LIN {X 0,Y 487.957,Z 631.751,A -85,B 0,C 180,E1 -6386.696,E2 -6386.696} C_VEL
LIN {X 0,Y 487.888,Z 633.791,A -85,B 0,C 180,E1 -6388.348,E2 -6388.348} C_VEL
LIN {X 0,Y 487.818,Z 634.497,A -85,B 0,C 180,E1 -6389.999,E2 -6389.999} C_VEL
LIN {X 0,Y 487.886,Z 633.877,A -85,B 0,C 180,E1 -6391.65,E2 -6391.65} C_VEL
LIN {X 0,Y 487.955,Z 631.916,A -85,B 0,C 180,E1 -6393.302,E2 -6393.302} C_VEL
LIN {X 0,Y 487.963,Z 628.565,A -85,B 0,C 180,E1 -6394.956,E2 -6394.956} C_VEL
LIN {X 0,Y 488.052,Z 624.185,A -85,B 0,C 180,E1 -6396.48,E2 -6396.48} C_VEL
LIN {X 0,Y 488.192,Z 619.062,A -85,B 0,C 180,E1 -6397.859,E2 -6397.859} C_VEL
LIN {X 0,Y 488.465,Z 612.281,A -85,B 0,C 180,E1 -6399.314,E2 -6399.314} C_VEL
LIN {X 0,Y 488.822,Z 603.853,A -85,B 0,C 180,E1 -6400.771,E2 -6400.771} C_VEL
LIN {X 0,Y 489.247,Z 594.601,A -85,B 0,C 180,E1 -6402.081,E2 -6402.081} C_VEL
LIN {X 0,Y 489.717,Z 584.411,A -85,B 0,C 180,E1 -6403.273,E2 -6403.273} C_VEL
LIN {X 0,Y 490.248,Z 573.643,A -85,B 0,C 180,E1 -6404.316,E2 -6404.316} C_VEL
LIN {X 0,Y 490.821,Z 561.869,A -85,B 0,C 180,E1 -6405.253,E2 -6405.253} C_VEL
LIN {X 0,Y 491.354,Z 548.87,A -85,B 0,C 180,E1 -6406.088,E2 -6406.088} C_VEL
LIN {X 0,Y 491.917,Z 535.085,A -85,B 0,C 180,E1 -6406.769,E2 -6406.769} C_VEL
LIN {X 0,Y 492.27,Z 521.352,A -85,B 0,C 180,E1 -6407.27,E2 -6407.27} C_VEL
LIN {X 0,Y 492.606,Z 506.72,A -85,B 0,C 180,E1 -6407.62,E2 -6407.62} C_VEL
LIN {X 0,Y 493.536,Z 388.715,A -85,B 0,C 180,E1 -6409.371,E2 -6409.371} C_VEL
LIN {X 0,Y 490.364,Z 372.401,A -85,B 0,C 180,E1 -6409.769,E2 -6409.769} C_VEL
LIN {X 0,Y 490.626,Z 364.751,A -85,B 0,C 180,E1 -6410.983,E2 -6410.983} C_VEL
LIN {X 0,Y 491.223,Z 351.672,A -85,B 0,C 180,E1 -6413.168,E2 -6413.168} C_VEL
LIN {X 0,Y 490.46,Z 346.443,A -85,B 0,C 180,E1 -6414.102,E2 -6414.102} C_VEL
LIN {X 0,Y 488.842,Z 338.631,A -85,B 0,C 180,E1 -6415.549,E2 -6415.549} C_VEL
LIN {X 0,Y 488.781,Z 338.212,A -85,B 0,C 180,E1 -6415.781,E2 -6415.781} C_VEL
LIN {X 0,Y 488.735,Z 338.214,A -85,B 0,C 180,E1 -6418.696,E2 -6418.696} C_VEL
LIN {X 0,Y 488.694,Z 338.234,A -85,B 0,C 180,E1 -6421.178,E2 -6421.178} C_VEL
LIN {X 0,Y 488.732,Z 338.235,A -85,B 0,C 180,E1 -6424.111,E2 -6424.111} C_VEL
LIN {X 0,Y 488.679,Z 338.234,A -85,B 0,C 180,E1 -6427.157,E2 -6427.157} C_VEL
LIN {X 0,Y 488.744,Z 338.225,A -85,B 0,C 180,E1 -6429.248,E2 -6429.248} C_VEL
LIN {X 0,Y 488.726,Z 338.23,A -85,B 0,C 180,E1 -6432.52,E2 -6432.52} C_VEL
LIN {X 0,Y 488.705,Z 338.222,A -85,B 0,C 180,E1 -6435.198,E2 -6435.198} C_VEL
LIN {X 0,Y 488.727,Z 338.229,A -85,B 0,C 180,E1 -6437.478,E2 -6437.478} C_VEL
LIN {X 0,Y 488.741,Z 338.22,A -85,B 0,C 180,E1 -6440.749,E2 -6440.749} C_VEL
LIN {X 0,Y 488.678,Z 338.232,A -85,B 0,C 180,E1 -6443.868,E2 -6443.868} C_VEL
LIN {X 0,Y 488.731,Z 338.229,A -85,B 0,C 180,E1 -6446.876,E2 -6446.876} C_VEL
LIN {X 0,Y 488.725,Z 338.215,A -85,B 0,C 180,E1 -6449.781,E2 -6449.781} C_VEL
LIN {X 0,Y 488.789,Z 338.211,A -85,B 0,C 180,E1 -6453.054,E2 -6453.054} C_VEL
LIN {X 0,Y 488.692,Z 338.233,A -85,B 0,C 180,E1 -6456.254,E2 -6456.254} C_VEL
LIN {X 0,Y 488.737,Z 338.225,A -85,B 0,C 180,E1 -6459.175,E2 -6459.175} C_VEL
LIN {X 0,Y 488.748,Z 338.229,A -85,B 0,C 180,E1 -6461.627,E2 -6461.627} C_VEL
LIN {X 0,Y 488.754,Z 338.221,A -85,B 0,C 180,E1 -6464.999,E2 -6464.999} C_VEL
LIN {X 0,Y 488.822,Z 338.215,A -85,B 0,C 180,E1 -6468.388,E2 -6468.388} C_VEL
LIN {X 0,Y 488.809,Z 338.217,A -85,B 0,C 180,E1 -6471.733,E2 -6471.733} C_VEL
LIN {X 0,Y 488.852,Z 338.211,A -85,B 0,C 180,E1 -6474.224,E2 -6474.224} C_VEL
LIN {X 0,Y 488.953,Z 338.199,A -85,B 0,C 180,E1 -6477.529,E2 -6477.529} C_VEL
LIN {X 0,Y 488.959,Z 338.199,A -85,B 0,C 180,E1 -6480,E2 -6480} C_VEL
LIN {X 0,Y 488.953,Z 338.199,A -85,B 0,C 180,E1 -6482.471,E2 -6482.471} C_VEL
LIN {X 0,Y 488.853,Z 338.212,A -85,B 0,C 180,E1 -6485.776,E2 -6485.776} C_VEL
LIN {X 0,Y 488.808,Z 338.217,A -85,B 0,C 180,E1 -6488.266,E2 -6488.266} C_VEL
LIN {X 0,Y 488.821,Z 338.214,A -85,B 0,C 180,E1 -6491.612,E2 -6491.612} C_VEL
LIN {X 0,Y 488.754,Z 338.221,A -85,B 0,C 180,E1 -6495.001,E2 -6495.001} C_VEL
LIN {X 0,Y 488.744,Z 338.229,A -85,B 0,C 180,E1 -6498.443,E2 -6498.443} C_VEL
LIN {X 0,Y 488.702,Z 338.228,A -85,B 0,C 180,E1 -6501.071,E2 -6501.071} C_VEL
LIN {X 0,Y 488.691,Z 338.232,A -85,B 0,C 180,E1 -6503.746,E2 -6503.746} C_VEL
LIN {X 0,Y 488.789,Z 338.211,A -85,B 0,C 180,E1 -6506.946,E2 -6506.946} C_VEL
LIN {X 0,Y 488.7,Z 338.219,A -85,B 0,C 180,E1 -6510.364,E2 -6510.364} C_VEL
LIN {X 0,Y 488.727,Z 338.228,A -85,B 0,C 180,E1 -6513.485,E2 -6513.485} C_VEL
LIN {X 0,Y 488.681,Z 338.228,A -85,B 0,C 180,E1 -6516.357,E2 -6516.357} C_VEL
LIN {X 0,Y 488.734,Z 338.22,A -85,B 0,C 180,E1 -6519.251,E2 -6519.251} C_VEL
LIN {X 0,Y 488.727,Z 338.229,A -85,B 0,C 180,E1 -6522.522,E2 -6522.522} C_VEL
LIN {X 0,Y 488.705,Z 338.221,A -85,B 0,C 180,E1 -6525.2,E2 -6525.2} C_VEL
LIN {X 0,Y 488.725,Z 338.23,A -85,B 0,C 180,E1 -6527.48,E2 -6527.48} C_VEL
LIN {X 0,Y 488.743,Z 338.225,A -85,B 0,C 180,E1 -6530.752,E2 -6530.752} C_VEL
LIN {X 0,Y 488.681,Z 338.235,A -85,B 0,C 180,E1 -6533.87,E2 -6533.87} C_VEL
LIN {X 0,Y 488.735,Z 338.225,A -85,B 0,C 180,E1 -6536.879,E2 -6536.879} C_VEL
LIN {X 0,Y 488.731,Z 338.223,A -85,B 0,C 180,E1 -6539.783,E2 -6539.783} C_VEL
LIN {X 0,Y 488.796,Z 338.225,A -85,B 0,C 180,E1 -6543.056,E2 -6543.056} C_VEL
LIN {X 0,Y 488.813,Z 338.303,A -85,B 0,C 180,E1 -6544.392,E2 -6544.392} C_VEL
LIN {X 0,Y 491.086,Z 349.656,A -85,B 0,C 180,E1 -6546.526,E2 -6546.526} C_VEL
LIN {X 0,Y 491.009,Z 356.638,A -85,B 0,C 180,E1 -6547.711,E2 -6547.711} C_VEL
LIN {X 0,Y 490.34,Z 372.125,A -85,B 0,C 180,E1 -6550.257,E2 -6550.257} C_VEL
LIN {X 0,Y 491.847,Z 380.023,A -85,B 0,C 180,E1 -6550.473,E2 -6550.473} C_VEL
LIN {X 0,Y 493.591,Z 389.526,A -85,B 0,C 180,E1 -6550.689,E2 -6550.689} C_VEL
LIN {X 0,Y 492.541,Z 509.938,A -85,B 0,C 180,E1 -6552.485,E2 -6552.485} C_VEL
LIN {X 0,Y 492.18,Z 524.147,A -85,B 0,C 180,E1 -6552.864,E2 -6552.864} C_VEL
LIN {X 0,Y 491.837,Z 537.72,A -85,B 0,C 180,E1 -6553.395,E2 -6553.395} C_VEL
LIN {X 0,Y 491.344,Z 549.891,A -85,B 0,C 180,E1 -6554.019,E2 -6554.019} C_VEL
LIN {X 0,Y 490.785,Z 562.69,A -85,B 0,C 180,E1 -6554.852,E2 -6554.852} C_VEL
LIN {X 0,Y 490.242,Z 574.318,A -85,B 0,C 180,E1 -6555.79,E2 -6555.79} C_VEL
LIN {X 0,Y 489.611,Z 585.946,A -85,B 0,C 180,E1 -6556.935,E2 -6556.935} C_VEL
LIN {X 0,Y 489.247,Z 595.237,A -85,B 0,C 180,E1 -6558.046,E2 -6558.046} C_VEL
LIN {X 0,Y 488.842,Z 603.563,A -85,B 0,C 180,E1 -6559.229,E2 -6559.229} C_VEL
LIN {X 0,Y 488.459,Z 612.04,A -85,B 0,C 180,E1 -6560.686,E2 -6560.686} C_VEL
LIN {X 0,Y 488.191,Z 618.866,A -85,B 0,C 180,E1 -6562.141,E2 -6562.141} C_VEL
LIN {X 0,Y 488.039,Z 624.895,A -85,B 0,C 180,E1 -6563.778,E2 -6563.778} C_VEL
LIN {X 0,Y 487.962,Z 628.449,A -85,B 0,C 180,E1 -6565.044,E2 -6565.044} C_VEL
LIN {X 0,Y 487.955,Z 631.837,A -85,B 0,C 180,E1 -6566.698,E2 -6566.698} C_VEL
LIN {X 0,Y 487.885,Z 633.838,A -85,B 0,C 180,E1 -6568.35,E2 -6568.35} C_VEL
LIN {X 0,Y 487.817,Z 634.5,A -85,B 0,C 180,E1 -6570.001,E2 -6570.001} C_VEL
LIN {X 0,Y 487.886,Z 633.834,A -85,B 0,C 180,E1 -6571.652,E2 -6571.652} C_VEL
LIN {X 0,Y 487.956,Z 631.83,A -85,B 0,C 180,E1 -6573.304,E2 -6573.304} C_VEL
LIN {X 0,Y 487.963,Z 628.441,A -85,B 0,C 180,E1 -6574.958,E2 -6574.958} C_VEL
LIN {X 0,Y 488.049,Z 624.037,A -85,B 0,C 180,E1 -6576.479,E2 -6576.479} C_VEL
LIN {X 0,Y 488.194,Z 618.859,A -85,B 0,C 180,E1 -6577.861,E2 -6577.861} C_VEL
LIN {X 0,Y 488.461,Z 612.028,A -85,B 0,C 180,E1 -6579.316,E2 -6579.316} C_VEL
LIN {X 0,Y 488.843,Z 603.549,A -85,B 0,C 180,E1 -6580.773,E2 -6580.773} C_VEL
LIN {X 0,Y 489.255,Z 594.224,A -85,B 0,C 180,E1 -6582.084,E2 -6582.084} C_VEL
LIN {X 0,Y 489.708,Z 583.976,A -85,B 0,C 180,E1 -6583.276,E2 -6583.276} C_VEL
LIN {X 0,Y 490.273,Z 573.121,A -85,B 0,C 180,E1 -6584.317,E2 -6584.317} C_VEL
LIN {X 0,Y 490.881,Z 561.232,A -85,B 0,C 180,E1 -6585.254,E2 -6585.254} C_VEL
LIN {X 0,Y 491.441,Z 548.081,A -85,B 0,C 180,E1 -6586.087,E2 -6586.087} C_VEL
LIN {X 0,Y 491.913,Z 534.836,A -85,B 0,C 180,E1 -6586.735,E2 -6586.735} C_VEL
LIN {X 0,Y 492.258,Z 520.818,A -85,B 0,C 180,E1 -6587.241,E2 -6587.241} C_VEL
LIN {X 0,Y 492.586,Z 507.071,A -85,B 0,C 180,E1 -6587.57,E2 -6587.57} C_VEL
LIN {X 0,Y 493.533,Z 389.002,A -85,B 0,C 180,E1 -6589.321,E2 -6589.321} C_VEL
LIN {X 0,Y 490.329,Z 372.216,A -85,B 0,C 180,E1 -6589.735,E2 -6589.735} C_VEL
LIN {X 0,Y 491.033,Z 355.31,A -85,B 0,C 180,E1 -6592.512,E2 -6592.512} C_VEL
LIN {X 0,Y 491.089,Z 349.648,A -85,B 0,C 180,E1 -6593.474,E2 -6593.474} C_VEL
LIN {X 0,Y 488.815,Z 338.438,A -85,B 0,C 180,E1 -6595.553,E2 -6595.553} C_VEL
LIN {X 0,Y 488.751,Z 338.231,A -85,B 0,C 180,E1 -6597.397,E2 -6597.397} C_VEL
LIN {X 0,Y 488.714,Z 338.236,A -85,B 0,C 180,E1 -6600.364,E2 -6600.364} C_VEL
LIN {X 0,Y 488.741,Z 338.229,A -85,B 0,C 180,E1 -6603.485,E2 -6603.485} C_VEL
LIN {X 0,Y 488.694,Z 338.238,A -85,B 0,C 180,E1 -6606.356,E2 -6606.356} C_VEL
LIN {X 0,Y 488.705,Z 338.233,A -85,B 0,C 180,E1 -6609.255,E2 -6609.255} C_VEL
LIN {X 0,Y 488.711,Z 338.234,A -85,B 0,C 180,E1 -6611.6,E2 -6611.6} C_VEL
LIN {X 0,Y 488.706,Z 338.231,A -85,B 0,C 180,E1 -6614.803,E2 -6614.803} C_VEL
LIN {X 0,Y 488.696,Z 338.237,A -85,B 0,C 180,E1 -6617.475,E2 -6617.475} C_VEL
LIN {X 0,Y 488.738,Z 338.233,A -85,B 0,C 180,E1 -6619.677,E2 -6619.677} C_VEL
LIN {X 0,Y 488.684,Z 338.236,A -85,B 0,C 180,E1 -6622.841,E2 -6622.841} C_VEL
LIN {X 0,Y 488.735,Z 338.234,A -85,B 0,C 180,E1 -6625.888,E2 -6625.888} C_VEL
LIN {X 0,Y 488.697,Z 338.236,A -85,B 0,C 180,E1 -6628.821,E2 -6628.821} C_VEL
LIN {X 0,Y 488.756,Z 338.232,A -85,B 0,C 180,E1 -6632.139,E2 -6632.139} C_VEL
LIN {X 0,Y 488.815,Z 338.538,A -85,B 0,C 180,E1 -6632.646,E2 -6632.646} C_VEL
LIN {X 0,Y 491.201,Z 350.219,A -85,B 0,C 180,E1 -6634.343,E2 -6634.343} C_VEL
LIN {X 0,Y 491.062,Z 365.26,A -85,B 0,C 180,E1 -6636.343,E2 -6636.343} C_VEL
LIN {X 0,Y 490.501,Z 386.847,A -85,B 0,C 180,E1 -6639.23,E2 -6639.23} C_VEL
LIN {X 0,Y 490.05,Z 409.49,A -85,B 0,C 180,E1 -6642.257,E2 -6642.257} C_VEL
LIN {X 0,Y 489.773,Z 420.832,A -85,B 0,C 180,E1 -6643.762,E2 -6643.762} C_VEL
LIN {X 0,Y 491.649,Z 435.316,A -85,B 0,C 180,E1 -6644.106,E2 -6644.106} C_VEL
LIN {X 0,Y 490.761,Z 532.213,A -85,B 0,C 180,E1 -6645.698,E2 -6645.698} C_VEL
LIN {X 0,Y 490.493,Z 544.73,A -85,B 0,C 180,E1 -6646.061,E2 -6646.061} C_VEL
LIN {X 0,Y 490.174,Z 557.03,A -85,B 0,C 180,E1 -6646.58,E2 -6646.58} C_VEL
LIN {X 0,Y 489.83,Z 569.483,A -85,B 0,C 180,E1 -6647.281,E2 -6647.281} C_VEL
LIN {X 0,Y 489.49,Z 580.545,A -85,B 0,C 180,E1 -6648.089,E2 -6648.089} C_VEL
LIN {X 0,Y 489.108,Z 590.871,A -85,B 0,C 180,E1 -6649.025,E2 -6649.025} C_VEL
LIN {X 0,Y 488.755,Z 600.216,A -85,B 0,C 180,E1 -6650.064,E2 -6650.064} C_VEL
LIN {X 0,Y 488.471,Z 609.197,A -85,B 0,C 180,E1 -6651.311,E2 -6651.311} C_VEL
LIN {X 0,Y 488.206,Z 616.433,A -85,B 0,C 180,E1 -6652.556,E2 -6652.556} C_VEL
LIN {X 0,Y 488.063,Z 622.035,A -85,B 0,C 180,E1 -6653.759,E2 -6653.759} C_VEL
LIN {X 0,Y 487.97,Z 626.714,A -85,B 0,C 180,E1 -6655.043,E2 -6655.043} C_VEL
LIN {X 0,Y 487.94,Z 629.073,A -85,B 0,C 180,E1 -6655.87,E2 -6655.87} C_VEL
LIN {X 0,Y 487.967,Z 631.002,A -85,B 0,C 180,E1 -6656.697,E2 -6656.697} C_VEL
LIN {X 0,Y 487.888,Z 632.494,A -85,B 0,C 180,E1 -6657.523,E2 -6657.523} C_VEL
LIN {X 0,Y 487.89,Z 633.528,A -85,B 0,C 180,E1 -6658.349,E2 -6658.349} C_VEL
LIN {X 0,Y 487.82,Z 634.417,A -85,B 0,C 180,E1 -6660,E2 -6660} C_VEL
LIN {X 0,Y 487.834,Z 634.223,A -85,B 0,C 180,E1 -6660.826,E2 -6660.826} C_VEL
LIN {X 0,Y 487.889,Z 633.621,A -85,B 0,C 180,E1 -6661.651,E2 -6661.651} C_VEL
LIN {X 0,Y 487.888,Z 632.625,A -85,B 0,C 180,E1 -6662.477,E2 -6662.477} C_VEL
LIN {X 0,Y 487.967,Z 631.209,A -85,B 0,C 180,E1 -6663.303,E2 -6663.303} C_VEL
LIN {X 0,Y 487.931,Z 628.245,A -85,B 0,C 180,E1 -6664.544,E2 -6664.544} C_VEL
LIN {X 0,Y 488.073,Z 624.216,A -85,B 0,C 180,E1 -6665.785,E2 -6665.785} C_VEL
LIN {X 0,Y 488.186,Z 618.005,A -85,B 0,C 180,E1 -6667.237,E2 -6667.237} C_VEL
LIN {X 0,Y 488.419,Z 611.228,A -85,B 0,C 180,E1 -6668.482,E2 -6668.482} C_VEL
LIN {X 0,Y 488.675,Z 602.725,A -85,B 0,C 180,E1 -6669.729,E2 -6669.729} C_VEL
LIN {X 0,Y 488.979,Z 594.009,A -85,B 0,C 180,E1 -6670.769,E2 -6670.769} C_VEL
LIN {X 0,Y 489.467,Z 583.309,A -85,B 0,C 180,E1 -6671.807,E2 -6671.807} C_VEL
LIN {X 0,Y 489.783,Z 572.519,A -85,B 0,C 180,E1 -6672.643,E2 -6672.643} C_VEL
LIN {X 0,Y 490.141,Z 560.667,A -85,B 0,C 180,E1 -6673.369,E2 -6673.369} C_VEL
LIN {X 0,Y 490.479,Z 548.288,A -85,B 0,C 180,E1 -6673.94,E2 -6673.94} C_VEL
LIN {X 0,Y 490.813,Z 534.532,A -85,B 0,C 180,E1 -6674.38,E2 -6674.38} C_VEL
LIN {X 0,Y 490.944,Z 519.124,A -85,B 0,C 180,E1 -6674.667,E2 -6674.667} C_VEL
LIN {X 0,Y 491.526,Z 433.033,A -85,B 0,C 180,E1 -6676.033,E2 -6676.033} C_VEL
LIN {X 0,Y 489.765,Z 420.903,A -85,B 0,C 180,E1 -6676.318,E2 -6676.318} C_VEL
LIN {X 0,Y 490.41,Z 396.325,A -85,B 0,C 180,E1 -6679.681,E2 -6679.681} C_VEL
LIN {X 0,Y 491.082,Z 374.245,A -85,B 0,C 180,E1 -6682.731,E2 -6682.731} C_VEL
LIN {X 0,Y 491.695,Z 353.431,A -85,B 0,C 180,E1 -6685.621,E2 -6685.621} C_VEL
LIN {X 0,Y 490.347,Z 345.54,A -85,B 0,C 180,E1 -6686.796,E2 -6686.796} C_VEL
LIN {X 0,Y 488.786,Z 338.35,A -85,B 0,C 180,E1 -6687.918,E2 -6687.918} C_VEL
LIN {X 0,Y 488.697,Z 338.235,A -85,B 0,C 180,E1 -6691.18,E2 -6691.18} C_VEL
LIN {X 0,Y 488.736,Z 338.233,A -85,B 0,C 180,E1 -6694.113,E2 -6694.113} C_VEL
LIN {X 0,Y 488.684,Z 338.234,A -85,B 0,C 180,E1 -6697.159,E2 -6697.159} C_VEL
LIN {X 0,Y 488.724,Z 338.235,A -85,B 0,C 180,E1 -6700.344,E2 -6700.344} C_VEL
LIN {X 0,Y 488.689,Z 338.232,A -85,B 0,C 180,E1 -6703.654,E2 -6703.654} C_VEL
LIN {X 0,Y 488.705,Z 338.222,A -85,B 0,C 180,E1 -6704.878,E2 -6704.878} C_VEL
LIN {X 0,Y 488.034,Z 338.306,A -85,B 0,C 180,E1 -6705.566,E2 -6705.566} C_VEL
LIN {X 0,Y 485.172,Z 338.674,A -85,B 0,C 180,E1 -6706.682,E2 -6706.682} C_VEL
LIN {X 0,Y 482.757,Z 338.978,A -85,B 0,C 180,E1 -6707.581,E2 -6707.581} C_VEL
LIN {X 0,Y 481.726,Z 339.105,A -85,B 0,C 180,E1 -6708.276,E2 -6708.276} C_VEL
LIN {X 0,Y 481.646,Z 339.112,A -85,B 0,C 180,E1 -6708.511,E2 -6708.511} C_VEL
LIN {X 0,Y 481.676,Z 339.104,A -85,B 0,C 180,E1 -6711.14,E2 -6711.14} C_VEL
LIN {X 0,Y 481.673,Z 339.107,A -85,B 0,C 180,E1 -6714.794,E2 -6714.794} C_VEL
LIN {X 0,Y 481.677,Z 339.106,A -85,B 0,C 180,E1 -6717.325,E2 -6717.325} C_VEL
LIN {X 0,Y 481.684,Z 339.093,A -85,B 0,C 180,E1 -6720.258,E2 -6720.258} C_VEL
LIN {X 0,Y 481.751,Z 339.101,A -85,B 0,C 180,E1 -6723.112,E2 -6723.112} C_VEL
LIN {X 0,Y 481.765,Z 339.248,A -85,B 0,C 180,E1 -6724.227,E2 -6724.227} C_VEL
LIN {X 0,Y 484.235,Z 351.61,A -85,B 0,C 180,E1 -6726.56,E2 -6726.56} C_VEL
LIN {X 0,Y 483.73,Z 365.505,A -85,B 0,C 180,E1 -6728.924,E2 -6728.924} C_VEL
LIN {X 0,Y 483.415,Z 372.218,A -85,B 0,C 180,E1 -6730.016,E2 -6730.016} C_VEL
LIN {X 0,Y 486.762,Z 389.518,A -85,B 0,C 180,E1 -6730.453,E2 -6730.453} C_VEL
LIN {X 0,Y 485.93,Z 499.574,A -85,B 0,C 180,E1 -6732.1,E2 -6732.1} C_VEL
LIN {X 0,Y 485.686,Z 515.129,A -85,B 0,C 180,E1 -6732.398,E2 -6732.398} C_VEL
LIN {X 0,Y 485.31,Z 528.714,A -85,B 0,C 180,E1 -6732.822,E2 -6732.822} C_VEL
LIN {X 0,Y 484.842,Z 542.31,A -85,B 0,C 180,E1 -6733.418,E2 -6733.418} C_VEL
LIN {X 0,Y 484.262,Z 555.958,A -85,B 0,C 180,E1 -6734.209,E2 -6734.209} C_VEL
LIN {X 0,Y 483.564,Z 568.872,A -85,B 0,C 180,E1 -6735.157,E2 -6735.157} C_VEL
LIN {X 0,Y 482.965,Z 580.493,A -85,B 0,C 180,E1 -6736.214,E2 -6736.214} C_VEL
LIN {X 0,Y 482.406,Z 591.008,A -85,B 0,C 180,E1 -6737.376,E2 -6737.376} C_VEL
LIN {X 0,Y 481.979,Z 600.501,A -85,B 0,C 180,E1 -6738.646,E2 -6738.646} C_VEL
LIN {X 0,Y 481.554,Z 609.56,A -85,B 0,C 180,E1 -6740.125,E2 -6740.125} C_VEL
LIN {X 0,Y 481.242,Z 616.857,A -85,B 0,C 180,E1 -6741.602,E2 -6741.602} C_VEL
LIN {X 0,Y 480.999,Z 623.414,A -85,B 0,C 180,E1 -6743.286,E2 -6743.286} C_VEL
LIN {X 0,Y 480.898,Z 628.327,A -85,B 0,C 180,E1 -6744.968,E2 -6744.968} C_VEL
LIN {X 0,Y 480.88,Z 631.752,A -85,B 0,C 180,E1 -6746.648,E2 -6746.648} C_VEL
LIN {X 0,Y 480.789,Z 633.792,A -85,B 0,C 180,E1 -6748.324,E2 -6748.324} C_VEL
LIN {X 0,Y 480.742,Z 634.497,A -85,B 0,C 180,E1 -6749.999,E2 -6749.999} C_VEL
LIN {X 0,Y 480.787,Z 633.876,A -85,B 0,C 180,E1 -6751.674,E2 -6751.674} C_VEL
LIN {X 0,Y 480.879,Z 631.915,A -85,B 0,C 180,E1 -6753.35,E2 -6753.35} C_VEL
LIN {X 0,Y 480.897,Z 628.563,A -85,B 0,C 180,E1 -6755.029,E2 -6755.029} C_VEL
LIN {X 0,Y 480.997,Z 623.723,A -85,B 0,C 180,E1 -6756.712,E2 -6756.712} C_VEL
LIN {X 0,Y 481.23,Z 617.251,A -85,B 0,C 180,E1 -6758.396,E2 -6758.396} C_VEL
LIN {X 0,Y 481.506,Z 610.046,A -85,B 0,C 180,E1 -6759.874,E2 -6759.874} C_VEL
LIN {X 0,Y 481.948,Z 601.134,A -85,B 0,C 180,E1 -6761.352,E2 -6761.352} C_VEL
LIN {X 0,Y 482.433,Z 591.777,A -85,B 0,C 180,E1 -6762.621,E2 -6762.621} C_VEL
LIN {X 0,Y 482.937,Z 581.412,A -85,B 0,C 180,E1 -6763.785,E2 -6763.785} C_VEL
LIN {X 0,Y 483.513,Z 569.982,A -85,B 0,C 180,E1 -6764.843,E2 -6764.843} C_VEL
LIN {X 0,Y 484.16,Z 557.317,A -85,B 0,C 180,E1 -6765.792,E2 -6765.792} C_VEL
LIN {X 0,Y 484.722,Z 544.996,A -85,B 0,C 180,E1 -6766.53,E2 -6766.53} C_VEL
LIN {X 0,Y 485.193,Z 531.363,A -85,B 0,C 180,E1 -6767.164,E2 -6767.164} C_VEL
LIN {X 0,Y 485.631,Z 517.184,A -85,B 0,C 180,E1 -6767.637,E2 -6767.637} C_VEL
LIN {X 0,Y 485.887,Z 503.683,A -85,B 0,C 180,E1 -6767.926,E2 -6767.926} C_VEL
LIN {X 0,Y 486.829,Z 389.653,A -85,B 0,C 180,E1 -6769.634,E2 -6769.634} C_VEL
LIN {X 0,Y 483.481,Z 372.451,A -85,B 0,C 180,E1 -6770.059,E2 -6770.059} C_VEL
LIN {X 0,Y 483.637,Z 367.364,A -85,B 0,C 180,E1 -6770.855,E2 -6770.855} C_VEL
LIN {X 0,Y 484.274,Z 352.055,A -85,B 0,C 180,E1 -6773.453,E2 -6773.453} C_VEL
LIN {X 0,Y 481.853,Z 339.681,A -85,B 0,C 180,E1 -6775.755,E2 -6775.755} C_VEL
LIN {X 0,Y 481.733,Z 339.118,A -85,B 0,C 180,E1 -6775.954,E2 -6775.954} C_VEL
LIN {X 0,Y 481.683,Z 339.09,A -85,B 0,C 180,E1 -6778.904,E2 -6778.904} C_VEL
LIN {X 0,Y 481.657,Z 339.111,A -85,B 0,C 180,E1 -6782.189,E2 -6782.189} C_VEL
LIN {X 0,Y 481.69,Z 339.106,A -85,B 0,C 180,E1 -6784.68,E2 -6784.68} C_VEL
LIN {X 0,Y 481.657,Z 339.116,A -85,B 0,C 180,E1 -6788.007,E2 -6788.007} C_VEL
LIN {X 0,Y 481.68,Z 339.104,A -85,B 0,C 180,E1 -6790.649,E2 -6790.649} C_VEL
LIN {X 0,Y 481.677,Z 339.108,A -85,B 0,C 180,E1 -6793.294,E2 -6793.294} C_VEL
LIN {X 0,Y 481.683,Z 339.102,A -85,B 0,C 180,E1 -6796.845,E2 -6796.845} C_VEL
LIN {X 0,Y 481.686,Z 339.103,A -85,B 0,C 180,E1 -6800.06,E2 -6800.06} C_VEL
LIN {X 0,Y 481.621,Z 339.101,A -85,B 0,C 180,E1 -6803.252,E2 -6803.252} C_VEL
LIN {X 0,Y 481.701,Z 339.105,A -85,B 0,C 180,E1 -6806.329,E2 -6806.329} C_VEL
LIN {X 0,Y 481.65,Z 339.101,A -85,B 0,C 180,E1 -6809.415,E2 -6809.415} C_VEL
LIN {X 0,Y 481.694,Z 339.093,A -85,B 0,C 180,E1 -6812.168,E2 -6812.168} C_VEL
LIN {X 0,Y 481.71,Z 339.102,A -85,B 0,C 180,E1 -6814.969,E2 -6814.969} C_VEL
LIN {X 0,Y 481.65,Z 339.109,A -85,B 0,C 180,E1 -6817.705,E2 -6817.705} C_VEL
LIN {X 0,Y 481.698,Z 339.102,A -85,B 0,C 180,E1 -6820.393,E2 -6820.393} C_VEL
LIN {X 0,Y 481.682,Z 339.109,A -85,B 0,C 180,E1 -6823.034,E2 -6823.034} C_VEL
LIN {X 0,Y 481.684,Z 339.107,A -85,B 0,C 180,E1 -6825.638,E2 -6825.638} C_VEL
LIN {X 0,Y 481.786,Z 339.091,A -85,B 0,C 180,E1 -6828.216,E2 -6828.216} C_VEL
LIN {X 0,Y 481.754,Z 339.097,A -85,B 0,C 180,E1 -6831.611,E2 -6831.611} C_VEL
LIN {X 0,Y 481.812,Z 339.088,A -85,B 0,C 180,E1 -6834.139,E2 -6834.139} C_VEL
LIN {X 0,Y 481.92,Z 339.076,A -85,B 0,C 180,E1 -6837.492,E2 -6837.492} C_VEL
LIN {X 0,Y 481.93,Z 339.075,A -85,B 0,C 180,E1 -6840,E2 -6840} C_VEL
LIN {X 0,Y 481.92,Z 339.075,A -85,B 0,C 180,E1 -6842.507,E2 -6842.507} C_VEL
LIN {X 0,Y 481.812,Z 339.088,A -85,B 0,C 180,E1 -6845.86,E2 -6845.86} C_VEL
LIN {X 0,Y 481.754,Z 339.096,A -85,B 0,C 180,E1 -6848.388,E2 -6848.388} C_VEL
LIN {X 0,Y 481.785,Z 339.09,A -85,B 0,C 180,E1 -6851.784,E2 -6851.784} C_VEL
LIN {X 0,Y 481.733,Z 339.093,A -85,B 0,C 180,E1 -6855.224,E2 -6855.224} C_VEL
LIN {X 0,Y 481.702,Z 339.108,A -85,B 0,C 180,E1 -6858.722,E2 -6858.722} C_VEL
LIN {X 0,Y 481.644,Z 339.105,A -85,B 0,C 180,E1 -6861.395,E2 -6861.395} C_VEL
LIN {X 0,Y 481.672,Z 339.109,A -85,B 0,C 180,E1 -6864.113,E2 -6864.113} C_VEL
LIN {X 0,Y 481.742,Z 339.087,A -85,B 0,C 180,E1 -6867.141,E2 -6867.141} C_VEL
LIN {X 0,Y 481.669,Z 339.087,A -85,B 0,C 180,E1 -6869.742,E2 -6869.742} C_VEL
LIN {X 0,Y 481.664,Z 339.113,A -85,B 0,C 180,E1 -6872.675,E2 -6872.675} C_VEL
LIN {X 0,Y 481.634,Z 339.11,A -85,B 0,C 180,E1 -6875.71,E2 -6875.71} C_VEL
LIN {X 0,Y 481.706,Z 339.096,A -85,B 0,C 180,E1 -6879.355,E2 -6879.355} C_VEL
LIN {X 0,Y 481.668,Z 339.114,A -85,B 0,C 180,E1 -6882.159,E2 -6882.159} C_VEL
LIN {X 0,Y 481.653,Z 339.101,A -85,B 0,C 180,E1 -6884.458,E2 -6884.458} C_VEL
LIN {X 0,Y 481.681,Z 339.107,A -85,B 0,C 180,E1 -6886.847,E2 -6886.847} C_VEL
LIN {X 0,Y 481.687,Z 339.103,A -85,B 0,C 180,E1 -6890.062,E2 -6890.062} C_VEL
LIN {X 0,Y 481.625,Z 339.113,A -85,B 0,C 180,E1 -6893.255,E2 -6893.255} C_VEL
LIN {X 0,Y 481.704,Z 339.104,A -85,B 0,C 180,E1 -6896.331,E2 -6896.331} C_VEL
LIN {X 0,Y 481.655,Z 339.112,A -85,B 0,C 180,E1 -6899.417,E2 -6899.417} C_VEL
LIN {X 0,Y 481.7,Z 339.103,A -85,B 0,C 180,E1 -6902.17,E2 -6902.17} C_VEL
LIN {X 0,Y 481.748,Z 339.162,A -85,B 0,C 180,E1 -6904.136,E2 -6904.136} C_VEL
LIN {X 0,Y 482.952,Z 344.873,A -85,B 0,C 180,E1 -6905.269,E2 -6905.269} C_VEL
LIN {X 0,Y 484.322,Z 352.933,A -85,B 0,C 180,E1 -6906.746,E2 -6906.746} C_VEL
LIN {X 0,Y 483.425,Z 372.023,A -85,B 0,C 180,E1 -6909.952,E2 -6909.952} C_VEL
LIN {X 0,Y 484.269,Z 376.511,A -85,B 0,C 180,E1 -6910.1,E2 -6910.1} C_VEL
LIN {X 0,Y 486.857,Z 389.883,A -85,B 0,C 180,E1 -6910.416,E2 -6910.416} C_VEL
LIN {X 0,Y 485.785,Z 509.946,A -85,B 0,C 180,E1 -6912.233,E2 -6912.233} C_VEL
LIN {X 0,Y 485.394,Z 524.487,A -85,B 0,C 180,E1 -6912.629,E2 -6912.629} C_VEL
LIN {X 0,Y 484.992,Z 538.853,A -85,B 0,C 180,E1 -6913.208,E2 -6913.208} C_VEL
LIN {X 0,Y 484.441,Z 551.66,A -85,B 0,C 180,E1 -6913.893,E2 -6913.893} C_VEL
LIN {X 0,Y 483.829,Z 564.118,A -85,B 0,C 180,E1 -6914.736,E2 -6914.736} C_VEL
LIN {X 0,Y 483.19,Z 576.663,A -85,B 0,C 180,E1 -6915.793,E2 -6915.793} C_VEL
LIN {X 0,Y 482.568,Z 587.841,A -85,B 0,C 180,E1 -6916.955,E2 -6916.955} C_VEL
LIN {X 0,Y 482.139,Z 597.86,A -85,B 0,C 180,E1 -6918.226,E2 -6918.226} C_VEL
LIN {X 0,Y 481.69,Z 606.18,A -85,B 0,C 180,E1 -6919.493,E2 -6919.493} C_VEL
LIN {X 0,Y 481.326,Z 614.132,A -85,B 0,C 180,E1 -6920.97,E2 -6920.97} C_VEL
LIN {X 0,Y 481.053,Z 620.53,A -85,B 0,C 180,E1 -6922.446,E2 -6922.446} C_VEL
LIN {X 0,Y 480.952,Z 626.204,A -85,B 0,C 180,E1 -6924.13,E2 -6924.13} C_VEL
LIN {X 0,Y 480.816,Z 630.322,A -85,B 0,C 180,E1 -6925.81,E2 -6925.81} C_VEL
LIN {X 0,Y 480.879,Z 631.837,A -85,B 0,C 180,E1 -6926.65,E2 -6926.65} C_VEL
LIN {X 0,Y 480.786,Z 633.838,A -85,B 0,C 180,E1 -6928.326,E2 -6928.326} C_VEL
LIN {X 0,Y 480.741,Z 634.5,A -85,B 0,C 180,E1 -6930.001,E2 -6930.001} C_VEL
LIN {X 0,Y 480.787,Z 633.834,A -85,B 0,C 180,E1 -6931.676,E2 -6931.676} C_VEL
LIN {X 0,Y 480.88,Z 631.83,A -85,B 0,C 180,E1 -6933.352,E2 -6933.352} C_VEL
LIN {X 0,Y 480.897,Z 628.441,A -85,B 0,C 180,E1 -6935.032,E2 -6935.032} C_VEL
LIN {X 0,Y 480.998,Z 623.565,A -85,B 0,C 180,E1 -6936.714,E2 -6936.714} C_VEL
LIN {X 0,Y 481.232,Z 617.05,A -85,B 0,C 180,E1 -6938.399,E2 -6938.399} C_VEL
LIN {X 0,Y 481.522,Z 609.797,A -85,B 0,C 180,E1 -6939.876,E2 -6939.876} C_VEL
LIN {X 0,Y 481.976,Z 600.815,A -85,B 0,C 180,E1 -6941.354,E2 -6941.354} C_VEL
LIN {X 0,Y 482.407,Z 591.383,A -85,B 0,C 180,E1 -6942.624,E2 -6942.624} C_VEL
LIN {X 0,Y 482.951,Z 580.941,A -85,B 0,C 180,E1 -6943.787,E2 -6943.787} C_VEL
LIN {X 0,Y 483.57,Z 569.411,A -85,B 0,C 180,E1 -6944.843,E2 -6944.843} C_VEL
LIN {X 0,Y 484.212,Z 556.617,A -85,B 0,C 180,E1 -6945.793,E2 -6945.793} C_VEL
LIN {X 0,Y 484.71,Z 544.128,A -85,B 0,C 180,E1 -6946.533,E2 -6946.533} C_VEL
LIN {X 0,Y 485.22,Z 531.003,A -85,B 0,C 180,E1 -6947.133,E2 -6947.133} C_VEL
LIN {X 0,Y 485.617,Z 517.779,A -85,B 0,C 180,E1 -6947.574,E2 -6947.574} C_VEL
LIN {X 0,Y 485.834,Z 504.051,A -85,B 0,C 180,E1 -6947.876,E2 -6947.876} C_VEL
LIN {X 0,Y 486.854,Z 390.543,A -85,B 0,C 180,E1 -6949.573,E2 -6949.573} C_VEL
LIN {X 0,Y 483.468,Z 372.591,A -85,B 0,C 180,E1 -6950.005,E2 -6950.005} C_VEL
LIN {X 0,Y 483.466,Z 370.871,A -85,B 0,C 180,E1 -6950.22,E2 -6950.22} C_VEL
LIN {X 0,Y 484.302,Z 352.912,A -85,B 0,C 180,E1 -6953.256,E2 -6953.256} C_VEL
LIN {X 0,Y 482.969,Z 344.846,A -85,B 0,C 180,E1 -6954.732,E2 -6954.732} C_VEL
LIN {X 0,Y 481.805,Z 339.393,A -85,B 0,C 180,E1 -6955.774,E2 -6955.774} C_VEL
LIN {X 0,Y 481.724,Z 339.096,A -85,B 0,C 180,E1 -6955.957,E2 -6955.957} C_VEL
LIN {X 0,Y 481.683,Z 339.095,A -85,B 0,C 180,E1 -6958.904,E2 -6958.904} C_VEL
LIN {X 0,Y 481.661,Z 339.116,A -85,B 0,C 180,E1 -6962.19,E2 -6962.19} C_VEL
LIN {X 0,Y 481.698,Z 339.107,A -85,B 0,C 180,E1 -6964.682,E2 -6964.682} C_VEL
LIN {X 0,Y 481.661,Z 339.114,A -85,B 0,C 180,E1 -6968.008,E2 -6968.008} C_VEL
LIN {X 0,Y 481.661,Z 339.109,A -85,B 0,C 180,E1 -6971.042,E2 -6971.042} C_VEL
LIN {X 0,Y 481.659,Z 339.111,A -85,B 0,C 180,E1 -6974.458,E2 -6974.458} C_VEL
LIN {X 0,Y 481.652,Z 339.115,A -85,B 0,C 180,E1 -6977.84,E2 -6977.84} C_VEL
LIN {X 0,Y 481.684,Z 339.107,A -85,B 0,C 180,E1 -6980.652,E2 -6980.652} C_VEL
LIN {X 0,Y 481.632,Z 339.118,A -85,B 0,C 180,E1 -6983.377,E2 -6983.377} C_VEL
LIN {X 0,Y 481.715,Z 339.106,A -85,B 0,C 180,E1 -6986.33,E2 -6986.33} C_VEL
LIN {X 0,Y 481.655,Z 339.116,A -85,B 0,C 180,E1 -6989.418,E2 -6989.418} C_VEL
LIN {X 0,Y 481.77,Z 339.27,A -85,B 0,C 180,E1 -6992.327,E2 -6992.327} C_VEL
LIN {X 0,Y 484.092,Z 350.058,A -85,B 0,C 180,E1 -6993.95,E2 -6993.95} C_VEL
LIN {X 0,Y 484.488,Z 355.178,A -85,B 0,C 180,E1 -6994.664,E2 -6994.664} C_VEL
LIN {X 0,Y 483.913,Z 379.969,A -85,B 0,C 180,E1 -6997.998,E2 -6997.998} C_VEL
LIN {X 0,Y 483.2,Z 404.701,A -85,B 0,C 180,E1 -7001.338,E2 -7001.338} C_VEL
LIN {X 0,Y 482.85,Z 420.811,A -85,B 0,C 180,E1 -7003.508,E2 -7003.508} C_VEL
LIN {X 0,Y 484.853,Z 436.091,A -85,B 0,C 180,E1 -7003.88,E2 -7003.88} C_VEL
LIN {X 0,Y 483.864,Z 531.429,A -85,B 0,C 180,E1 -7005.49,E2 -7005.49} C_VEL
LIN {X 0,Y 483.591,Z 544.231,A -85,B 0,C 180,E1 -7005.857,E2 -7005.857} C_VEL
LIN {X 0,Y 483.261,Z 556.641,A -85,B 0,C 180,E1 -7006.384,E2 -7006.384} C_VEL
LIN {X 0,Y 482.88,Z 569.273,A -85,B 0,C 180,E1 -7007.102,E2 -7007.102} C_VEL
LIN {X 0,Y 482.504,Z 580.282,A -85,B 0,C 180,E1 -7007.914,E2 -7007.914} C_VEL
LIN {X 0,Y 482.112,Z 590.645,A -85,B 0,C 180,E1 -7008.863,E2 -7008.863} C_VEL
LIN {X 0,Y 481.715,Z 600.03,A -85,B 0,C 180,E1 -7009.917,E2 -7009.917} C_VEL
LIN {X 0,Y 481.428,Z 609.061,A -85,B 0,C 180,E1 -7011.183,E2 -7011.183} C_VEL
LIN {X 0,Y 481.161,Z 616.33,A -85,B 0,C 180,E1 -7012.446,E2 -7012.446} C_VEL
LIN {X 0,Y 480.969,Z 622.43,A -85,B 0,C 180,E1 -7013.784,E2 -7013.784} C_VEL
LIN {X 0,Y 480.905,Z 626.663,A -85,B 0,C 180,E1 -7014.97,E2 -7014.97} C_VEL
LIN {X 0,Y 480.839,Z 629.033,A -85,B 0,C 180,E1 -7015.809,E2 -7015.809} C_VEL
LIN {X 0,Y 480.891,Z 630.97,A -85,B 0,C 180,E1 -7016.649,E2 -7016.649} C_VEL
LIN {X 0,Y 480.805,Z 632.471,A -85,B 0,C 180,E1 -7017.487,E2 -7017.487} C_VEL
LIN {X 0,Y 480.791,Z 633.51,A -85,B 0,C 180,E1 -7018.325,E2 -7018.325} C_VEL
LIN {X 0,Y 480.761,Z 634.154,A -85,B 0,C 180,E1 -7019.162,E2 -7019.162} C_VEL
LIN {X 0,Y 480.743,Z 634.404,A -85,B 0,C 180,E1 -7020,E2 -7020} C_VEL
LIN {X 0,Y 480.761,Z 634.208,A -85,B 0,C 180,E1 -7020.838,E2 -7020.838} C_VEL
LIN {X 0,Y 480.79,Z 633.601,A -85,B 0,C 180,E1 -7021.675,E2 -7021.675} C_VEL
LIN {X 0,Y 480.804,Z 632.601,A -85,B 0,C 180,E1 -7022.513,E2 -7022.513} C_VEL
LIN {X 0,Y 480.891,Z 631.175,A -85,B 0,C 180,E1 -7023.351,E2 -7023.351} C_VEL
LIN {X 0,Y 480.848,Z 628.196,A -85,B 0,C 180,E1 -7024.611,E2 -7024.611} C_VEL
LIN {X 0,Y 480.991,Z 624.145,A -85,B 0,C 180,E1 -7025.871,E2 -7025.871} C_VEL
LIN {X 0,Y 481.115,Z 617.905,A -85,B 0,C 180,E1 -7027.344,E2 -7027.344} C_VEL
LIN {X 0,Y 481.359,Z 611.099,A -85,B 0,C 180,E1 -7028.607,E2 -7028.607} C_VEL
LIN {X 0,Y 481.65,Z 602.544,A -85,B 0,C 180,E1 -7029.872,E2 -7029.872} C_VEL
LIN {X 0,Y 481.98,Z 593.783,A -85,B 0,C 180,E1 -7030.927,E2 -7030.927} C_VEL
LIN {X 0,Y 482.483,Z 583.019,A -85,B 0,C 180,E1 -7031.979,E2 -7031.979} C_VEL
LIN {X 0,Y 482.829,Z 571.579,A -85,B 0,C 180,E1 -7032.867,E2 -7032.867} C_VEL
LIN {X 0,Y 483.239,Z 559.206,A -85,B 0,C 180,E1 -7033.617,E2 -7033.617} C_VEL
LIN {X 0,Y 483.627,Z 546.24,A -85,B 0,C 180,E1 -7034.195,E2 -7034.195} C_VEL
LIN {X 0,Y 483.928,Z 533.62,A -85,B 0,C 180,E1 -7034.589,E2 -7034.589} C_VEL
LIN {X 0,Y 484.141,Z 512.741,A -85,B 0,C 180,E1 -7034.959,E2 -7034.959} C_VEL
LIN {X 0,Y 484.714,Z 434.014,A -85,B 0,C 180,E1 -7036.236,E2 -7036.236} C_VEL
LIN {X 0,Y 482.792,Z 420.858,A -85,B 0,C 180,E1 -7036.549,E2 -7036.549} C_VEL
LIN {X 0,Y 483.456,Z 397.671,A -85,B 0,C 180,E1 -7039.754,E2 -7039.754} C_VEL
LIN {X 0,Y 484.238,Z 373.88,A -85,B 0,C 180,E1 -7043.071,E2 -7043.071} C_VEL
LIN {X 0,Y 484.804,Z 354.557,A -85,B 0,C 180,E1 -7045.779,E2 -7045.779} C_VEL
LIN {X 0,Y 482.797,Z 343.949,A -85,B 0,C 180,E1 -7047.38,E2 -7047.38} C_VEL
LIN {X 0,Y 481.759,Z 339.208,A -85,B 0,C 180,E1 -7048.154,E2 -7048.154} C_VEL
LIN {X 0,Y 481.651,Z 339.117,A -85,B 0,C 180,E1 -7050.711,E2 -7050.711} C_VEL
LIN {X 0,Y 481.703,Z 339.106,A -85,B 0,C 180,E1 -7053.733,E2 -7053.733} C_VEL
LIN {X 0,Y 481.631,Z 339.116,A -85,B 0,C 180,E1 -7056.747,E2 -7056.747} C_VEL
LIN {X 0,Y 481.682,Z 339.11,A -85,B 0,C 180,E1 -7059.94,E2 -7059.94} C_VEL
LIN {X 0,Y 481.637,Z 339.109,A -85,B 0,C 180,E1 -7063.147,E2 -7063.147} C_VEL
LIN {X 0,Y 481.659,Z 339.1,A -85,B 0,C 180,E1 -7065.641,E2 -7065.641} C_VEL
LIN {X 0,Y 481.646,Z 339.112,A -85,B 0,C 180,E1 -7068.511,E2 -7068.511} C_VEL
LIN {X 0,Y 480.986,Z 339.191,A -85,B 0,C 180,E1 -7069.209,E2 -7069.209} C_VEL
LIN {X 0,Y 478.133,Z 339.545,A -85,B 0,C 180,E1 -7070.342,E2 -7070.342} C_VEL
LIN {X 0,Y 475.714,Z 339.848,A -85,B 0,C 180,E1 -7071.255,E2 -7071.255} C_VEL
LIN {X 0,Y 474.675,Z 339.983,A -85,B 0,C 180,E1 -7071.96,E2 -7071.96} C_VEL
LIN {X 0,Y 474.591,Z 339.989,A -85,B 0,C 180,E1 -7072.199,E2 -7072.199} C_VEL
LIN {X 0,Y 474.634,Z 339.984,A -85,B 0,C 180,E1 -7074.726,E2 -7074.726} C_VEL
LIN {X 0,Y 474.641,Z 339.984,A -85,B 0,C 180,E1 -7077.787,E2 -7077.787} C_VEL
LIN {X 0,Y 474.629,Z 339.968,A -85,B 0,C 180,E1 -7080.884,E2 -7080.884} C_VEL
LIN {X 0,Y 474.702,Z 340.015,A -85,B 0,C 180,E1 -7083.923,E2 -7083.923} C_VEL
LIN {X 0,Y 475.206,Z 342.399,A -85,B 0,C 180,E1 -7084.443,E2 -7084.443} C_VEL
LIN {X 0,Y 477.386,Z 353.743,A -85,B 0,C 180,E1 -7086.578,E2 -7086.578} C_VEL
LIN {X 0,Y 476.578,Z 371.201,A -85,B 0,C 180,E1 -7089.576,E2 -7089.576} C_VEL
LIN {X 0,Y 476.609,Z 372.727,A -85,B 0,C 180,E1 -7089.744,E2 -7089.744} C_VEL
LIN {X 0,Y 480.174,Z 391.553,A -85,B 0,C 180,E1 -7090.204,E2 -7090.204} C_VEL
LIN {X 0,Y 479.067,Z 509.07,A -85,B 0,C 180,E1 -7092.001,E2 -7092.001} C_VEL
LIN {X 0,Y 478.691,Z 523.172,A -85,B 0,C 180,E1 -7092.375,E2 -7092.375} C_VEL
LIN {X 0,Y 478.223,Z 537.604,A -85,B 0,C 180,E1 -7092.948,E2 -7092.948} C_VEL
LIN {X 0,Y 477.673,Z 550.894,A -85,B 0,C 180,E1 -7093.656,E2 -7093.656} C_VEL
LIN {X 0,Y 477.036,Z 563.493,A -85,B 0,C 180,E1 -7094.511,E2 -7094.511} C_VEL
LIN {X 0,Y 476.393,Z 574.981,A -85,B 0,C 180,E1 -7095.475,E2 -7095.475} C_VEL
LIN {X 0,Y 475.742,Z 585.52,A -85,B 0,C 180,E1 -7096.545,E2 -7096.545} C_VEL
LIN {X 0,Y 475.248,Z 595.855,A -85,B 0,C 180,E1 -7097.816,E2 -7097.816} C_VEL
LIN {X 0,Y 474.746,Z 604.62,A -85,B 0,C 180,E1 -7099.119,E2 -7099.119} C_VEL
LIN {X 0,Y 474.34,Z 612.898,A -85,B 0,C 180,E1 -7100.619,E2 -7100.619} C_VEL
LIN {X 0,Y 474.09,Z 618.668,A -85,B 0,C 180,E1 -7101.903,E2 -7101.903} C_VEL
LIN {X 0,Y 473.886,Z 624.597,A -85,B 0,C 180,E1 -7103.54,E2 -7103.54} C_VEL
LIN {X 0,Y 473.833,Z 628.328,A -85,B 0,C 180,E1 -7104.893,E2 -7104.893} C_VEL
LIN {X 0,Y 473.788,Z 631.753,A -85,B 0,C 180,E1 -7106.597,E2 -7106.597} C_VEL
LIN {X 0,Y 473.694,Z 633.792,A -85,B 0,C 180,E1 -7108.299,E2 -7108.299} C_VEL
LIN {X 0,Y 473.668,Z 634.497,A -85,B 0,C 180,E1 -7109.999,E2 -7109.999} C_VEL
LIN {X 0,Y 473.692,Z 633.876,A -85,B 0,C 180,E1 -7111.699,E2 -7111.699} C_VEL
LIN {X 0,Y 473.787,Z 631.914,A -85,B 0,C 180,E1 -7113.401,E2 -7113.401} C_VEL
LIN {X 0,Y 473.832,Z 628.562,A -85,B 0,C 180,E1 -7115.105,E2 -7115.105} C_VEL
LIN {X 0,Y 473.908,Z 623.721,A -85,B 0,C 180,E1 -7116.812,E2 -7116.812} C_VEL
LIN {X 0,Y 474.159,Z 617.248,A -85,B 0,C 180,E1 -7118.523,E2 -7118.523} C_VEL
LIN {X 0,Y 474.464,Z 610.043,A -85,B 0,C 180,E1 -7120.022,E2 -7120.022} C_VEL
LIN {X 0,Y 474.957,Z 601.131,A -85,B 0,C 180,E1 -7121.522,E2 -7121.522} C_VEL
LIN {X 0,Y 475.457,Z 591.773,A -85,B 0,C 180,E1 -7122.809,E2 -7122.809} C_VEL
LIN {X 0,Y 476.024,Z 581.407,A -85,B 0,C 180,E1 -7123.989,E2 -7123.989} C_VEL
LIN {X 0,Y 476.633,Z 569.976,A -85,B 0,C 180,E1 -7125.062,E2 -7125.062} C_VEL
LIN {X 0,Y 477.321,Z 557.31,A -85,B 0,C 180,E1 -7126.025,E2 -7126.025} C_VEL
LIN {X 0,Y 477.904,Z 545.321,A -85,B 0,C 180,E1 -7126.755,E2 -7126.755} C_VEL
LIN {X 0,Y 478.429,Z 531.351,A -85,B 0,C 180,E1 -7127.414,E2 -7127.414} C_VEL
LIN {X 0,Y 478.842,Z 518.084,A -85,B 0,C 180,E1 -7127.868,E2 -7127.868} C_VEL
LIN {X 0,Y 479.16,Z 503.657,A -85,B 0,C 180,E1 -7128.187,E2 -7128.187} C_VEL
LIN {X 0,Y 480.18,Z 390.809,A -85,B 0,C 180,E1 -7129.899,E2 -7129.899} C_VEL
LIN {X 0,Y 476.608,Z 372.566,A -85,B 0,C 180,E1 -7130.356,E2 -7130.356} C_VEL
LIN {X 0,Y 476.572,Z 371.83,A -85,B 0,C 180,E1 -7130.422,E2 -7130.422} C_VEL
LIN {X 0,Y 477.423,Z 354.282,A -85,B 0,C 180,E1 -7133.418,E2 -7133.418} C_VEL
LIN {X 0,Y 476.042,Z 346.435,A -85,B 0,C 180,E1 -7134.881,E2 -7134.881} C_VEL
LIN {X 0,Y 474.705,Z 340.096,A -85,B 0,C 180,E1 -7136.139,E2 -7136.139} C_VEL
LIN {X 0,Y 474.648,Z 339.973,A -85,B 0,C 180,E1 -7138.281,E2 -7138.281} C_VEL
LIN {X 0,Y 474.6,Z 339.991,A -85,B 0,C 180,E1 -7141.216,E2 -7141.216} C_VEL
LIN {X 0,Y 474.631,Z 339.99,A -85,B 0,C 180,E1 -7144.239,E2 -7144.239} C_VEL
LIN {X 0,Y 474.59,Z 339.991,A -85,B 0,C 180,E1 -7147.382,E2 -7147.382} C_VEL
LIN {X 0,Y 474.65,Z 339.979,A -85,B 0,C 180,E1 -7149.65,E2 -7149.65} C_VEL
LIN {X 0,Y 474.645,Z 339.983,A -85,B 0,C 180,E1 -7152.929,E2 -7152.929} C_VEL
LIN {X 0,Y 474.612,Z 339.98,A -85,B 0,C 180,E1 -7155.895,E2 -7155.895} C_VEL
LIN {X 0,Y 474.64,Z 339.984,A -85,B 0,C 180,E1 -7159.037,E2 -7159.037} C_VEL
LIN {X 0,Y 474.612,Z 339.974,A -85,B 0,C 180,E1 -7161.701,E2 -7161.701} C_VEL
LIN {X 0,Y 474.622,Z 339.983,A -85,B 0,C 180,E1 -7164.725,E2 -7164.725} C_VEL
LIN {X 0,Y 474.629,Z 339.985,A -85,B 0,C 180,E1 -7167.787,E2 -7167.787} C_VEL
LIN {X 0,Y 474.623,Z 339.964,A -85,B 0,C 180,E1 -7170.882,E2 -7170.882} C_VEL
LIN {X 0,Y 474.658,Z 339.978,A -85,B 0,C 180,E1 -7173.628,E2 -7173.628} C_VEL
LIN {X 0,Y 474.626,Z 339.985,A -85,B 0,C 180,E1 -7176.64,E2 -7176.64} C_VEL
LIN {X 0,Y 474.647,Z 339.981,A -85,B 0,C 180,E1 -7180.089,E2 -7180.089} C_VEL
LIN {X 0,Y 474.641,Z 339.983,A -85,B 0,C 180,E1 -7182.774,E2 -7182.774} C_VEL
LIN {X 0,Y 474.642,Z 339.983,A -85,B 0,C 180,E1 -7185.421,E2 -7185.421} C_VEL
LIN {X 0,Y 474.729,Z 339.97,A -85,B 0,C 180,E1 -7188.038,E2 -7188.038} C_VEL
LIN {X 0,Y 474.719,Z 339.974,A -85,B 0,C 180,E1 -7191.486,E2 -7191.486} C_VEL
LIN {X 0,Y 474.774,Z 339.965,A -85,B 0,C 180,E1 -7194.052,E2 -7194.052} C_VEL
LIN {X 0,Y 474.886,Z 339.952,A -85,B 0,C 180,E1 -7197.455,E2 -7197.455} C_VEL
LIN {X 0,Y 474.901,Z 339.95,A -85,B 0,C 180,E1 -7200,E2 -7200} C_VEL
LIN {X 0,Y 474.886,Z 339.951,A -85,B 0,C 180,E1 -7202.545,E2 -7202.545} C_VEL
LIN {X 0,Y 474.774,Z 339.965,A -85,B 0,C 180,E1 -7205.948,E2 -7205.948} C_VEL
LIN {X 0,Y 474.719,Z 339.974,A -85,B 0,C 180,E1 -7208.514,E2 -7208.514} C_VEL
LIN {X 0,Y 474.729,Z 339.97,A -85,B 0,C 180,E1 -7211.962,E2 -7211.962} C_VEL
LIN {X 0,Y 474.67,Z 339.97,A -85,B 0,C 180,E1 -7215.768,E2 -7215.768} C_VEL
LIN {X 0,Y 474.655,Z 339.982,A -85,B 0,C 180,E1 -7219.011,E2 -7219.011} C_VEL
LIN {X 0,Y 474.587,Z 339.983,A -85,B 0,C 180,E1 -7221.729,E2 -7221.729} C_VEL
LIN {X 0,Y 474.652,Z 339.988,A -85,B 0,C 180,E1 -7224.493,E2 -7224.493} C_VEL
LIN {X 0,Y 474.689,Z 339.964,A -85,B 0,C 180,E1 -7227.339,E2 -7227.339} C_VEL
LIN {X 0,Y 474.596,Z 339.983,A -85,B 0,C 180,E1 -7230.811,E2 -7230.811} C_VEL
LIN {X 0,Y 474.629,Z 339.988,A -85,B 0,C 180,E1 -7233.985,E2 -7233.985} C_VEL
LIN {X 0,Y 474.566,Z 339.978,A -85,B 0,C 180,E1 -7236.901,E2 -7236.901} C_VEL
LIN {X 0,Y 474.643,Z 339.977,A -85,B 0,C 180,E1 -7239.652,E2 -7239.652} C_VEL
LIN {X 0,Y 474.645,Z 339.98,A -85,B 0,C 180,E1 -7242.931,E2 -7242.931} C_VEL
LIN {X 0,Y 474.611,Z 339.981,A -85,B 0,C 180,E1 -7245.897,E2 -7245.897} C_VEL
LIN {X 0,Y 474.639,Z 339.98,A -85,B 0,C 180,E1 -7249.039,E2 -7249.039} C_VEL
LIN {X 0,Y 474.614,Z 339.988,A -85,B 0,C 180,E1 -7251.704,E2 -7251.704} C_VEL
LIN {X 0,Y 474.626,Z 339.985,A -85,B 0,C 180,E1 -7254.727,E2 -7254.727} C_VEL
LIN {X 0,Y 474.634,Z 339.985,A -85,B 0,C 180,E1 -7257.789,E2 -7257.789} C_VEL
LIN {X 0,Y 474.628,Z 339.967,A -85,B 0,C 180,E1 -7260.884,E2 -7260.884} C_VEL
LIN {X 0,Y 474.674,Z 339.972,A -85,B 0,C 180,E1 -7263.631,E2 -7263.631} C_VEL
LIN {X 0,Y 474.709,Z 340.13,A -85,B 0,C 180,E1 -7263.923,E2 -7263.923} C_VEL
LIN {X 0,Y 477.275,Z 352.897,A -85,B 0,C 180,E1 -7266.376,E2 -7266.376} C_VEL
LIN {X 0,Y 477.181,Z 359.256,A -85,B 0,C 180,E1 -7267.486,E2 -7267.486} C_VEL
LIN {X 0,Y 476.57,Z 372.244,A -85,B 0,C 180,E1 -7269.671,E2 -7269.671} C_VEL
LIN {X 0,Y 480.184,Z 391.631,A -85,B 0,C 180,E1 -7270.159,E2 -7270.159} C_VEL
LIN {X 0,Y 479.029,Z 509.955,A -85,B 0,C 180,E1 -7271.974,E2 -7271.974} C_VEL
LIN {X 0,Y 478.623,Z 524.425,A -85,B 0,C 180,E1 -7272.373,E2 -7272.373} C_VEL
LIN {X 0,Y 478.264,Z 537.728,A -85,B 0,C 180,E1 -7272.91,E2 -7272.91} C_VEL
LIN {X 0,Y 477.677,Z 549.932,A -85,B 0,C 180,E1 -7273.551,E2 -7273.551} C_VEL
LIN {X 0,Y 477.056,Z 562.695,A -85,B 0,C 180,E1 -7274.405,E2 -7274.405} C_VEL
LIN {X 0,Y 476.398,Z 574.321,A -85,B 0,C 180,E1 -7275.368,E2 -7275.368} C_VEL
LIN {X 0,Y 475.73,Z 585.948,A -85,B 0,C 180,E1 -7276.547,E2 -7276.547} C_VEL
LIN {X 0,Y 475.232,Z 596.207,A -85,B 0,C 180,E1 -7277.817,E2 -7277.817} C_VEL
LIN {X 0,Y 474.744,Z 604.918,A -85,B 0,C 180,E1 -7279.121,E2 -7279.121} C_VEL
LIN {X 0,Y 474.323,Z 613.126,A -85,B 0,C 180,E1 -7280.621,E2 -7280.621} C_VEL
LIN {X 0,Y 474.079,Z 618.867,A -85,B 0,C 180,E1 -7281.905,E2 -7281.905} C_VEL
LIN {X 0,Y 473.925,Z 624.602,A -85,B 0,C 180,E1 -7283.498,E2 -7283.498} C_VEL
LIN {X 0,Y 473.83,Z 628.449,A -85,B 0,C 180,E1 -7284.895,E2 -7284.895} C_VEL
LIN {X 0,Y 473.786,Z 631.837,A -85,B 0,C 180,E1 -7286.599,E2 -7286.599} C_VEL
LIN {X 0,Y 473.692,Z 633.838,A -85,B 0,C 180,E1 -7288.301,E2 -7288.301} C_VEL
LIN {X 0,Y 473.668,Z 634.5,A -85,B 0,C 180,E1 -7290.001,E2 -7290.001} C_VEL
LIN {X 0,Y 473.692,Z 633.834,A -85,B 0,C 180,E1 -7291.701,E2 -7291.701} C_VEL
LIN {X 0,Y 473.787,Z 631.829,A -85,B 0,C 180,E1 -7293.403,E2 -7293.403} C_VEL
LIN {X 0,Y 473.831,Z 628.44,A -85,B 0,C 180,E1 -7295.107,E2 -7295.107} C_VEL
LIN {X 0,Y 473.909,Z 623.565,A -85,B 0,C 180,E1 -7296.815,E2 -7296.815} C_VEL
LIN {X 0,Y 474.163,Z 617.049,A -85,B 0,C 180,E1 -7298.525,E2 -7298.525} C_VEL
LIN {X 0,Y 474.479,Z 609.796,A -85,B 0,C 180,E1 -7300.024,E2 -7300.024} C_VEL
LIN {X 0,Y 474.985,Z 600.814,A -85,B 0,C 180,E1 -7301.523,E2 -7301.523} C_VEL
LIN {X 0,Y 475.457,Z 591.381,A -85,B 0,C 180,E1 -7302.811,E2 -7302.811} C_VEL
LIN {X 0,Y 476.044,Z 580.939,A -85,B 0,C 180,E1 -7303.991,E2 -7303.991} C_VEL
LIN {X 0,Y 476.688,Z 569.409,A -85,B 0,C 180,E1 -7305.062,E2 -7305.062} C_VEL
LIN {X 0,Y 477.369,Z 556.614,A -85,B 0,C 180,E1 -7306.025,E2 -7306.025} C_VEL
LIN {X 0,Y 477.897,Z 544.299,A -85,B 0,C 180,E1 -7306.766,E2 -7306.766} C_VEL
LIN {X 0,Y 478.43,Z 531,A -85,B 0,C 180,E1 -7307.383,E2 -7307.383} C_VEL
LIN {X 0,Y 478.845,Z 517.772,A -85,B 0,C 180,E1 -7307.831,E2 -7307.831} C_VEL
LIN {X 0,Y 479.103,Z 504.04,A -85,B 0,C 180,E1 -7308.136,E2 -7308.136} C_VEL
LIN {X 0,Y 480.158,Z 391.387,A -85,B 0,C 180,E1 -7309.844,E2 -7309.844} C_VEL
LIN {X 0,Y 476.597,Z 372.607,A -85,B 0,C 180,E1 -7310.305,E2 -7310.305} C_VEL
LIN {X 0,Y 476.597,Z 370.87,A -85,B 0,C 180,E1 -7310.524,E2 -7310.524} C_VEL
LIN {X 0,Y 477.404,Z 354,A -85,B 0,C 180,E1 -7313.421,E2 -7313.421} C_VEL
LIN {X 0,Y 475.436,Z 343.536,A -85,B 0,C 180,E1 -7315.385,E2 -7315.385} C_VEL
LIN {X 0,Y 474.684,Z 340.012,A -85,B 0,C 180,E1 -7316.125,E2 -7316.125} C_VEL
LIN {X 0,Y 474.628,Z 339.974,A -85,B 0,C 180,E1 -7319.116,E2 -7319.116} C_VEL
LIN {X 0,Y 474.62,Z 339.99,A -85,B 0,C 180,E1 -7322.431,E2 -7322.431} C_VEL
LIN {X 0,Y 474.625,Z 339.989,A -85,B 0,C 180,E1 -7325.471,E2 -7325.471} C_VEL
LIN {X 0,Y 474.616,Z 339.99,A -85,B 0,C 180,E1 -7328.458,E2 -7328.458} C_VEL
LIN {X 0,Y 474.632,Z 339.985,A -85,B 0,C 180,E1 -7330.96,E2 -7330.96} C_VEL
LIN {X 0,Y 474.609,Z 339.991,A -85,B 0,C 180,E1 -7334.106,E2 -7334.106} C_VEL
LIN {X 0,Y 474.619,Z 339.988,A -85,B 0,C 180,E1 -7337.066,E2 -7337.066} C_VEL
LIN {X 0,Y 474.649,Z 339.985,A -85,B 0,C 180,E1 -7340.455,E2 -7340.455} C_VEL
LIN {X 0,Y 474.593,Z 339.995,A -85,B 0,C 180,E1 -7343.677,E2 -7343.677} C_VEL
LIN {X 0,Y 474.648,Z 339.986,A -85,B 0,C 180,E1 -7346.78,E2 -7346.78} C_VEL
LIN {X 0,Y 474.61,Z 339.995,A -85,B 0,C 180,E1 -7349.77,E2 -7349.77} C_VEL
LIN {X 0,Y 474.706,Z 340.188,A -85,B 0,C 180,E1 -7352.041,E2 -7352.041} C_VEL
LIN {X 0,Y 477.246,Z 351.601,A -85,B 0,C 180,E1 -7353.782,E2 -7353.782} C_VEL
LIN {X 0,Y 477.708,Z 356.962,A -85,B 0,C 180,E1 -7354.538,E2 -7354.538} C_VEL
LIN {X 0,Y 477.019,Z 381.581,A -85,B 0,C 180,E1 -7357.904,E2 -7357.904} C_VEL
LIN {X 0,Y 476.296,Z 406.388,A -85,B 0,C 180,E1 -7361.281,E2 -7361.281} C_VEL
LIN {X 0,Y 475.957,Z 420.933,A -85,B 0,C 180,E1 -7363.242,E2 -7363.242} C_VEL
LIN {X 0,Y 478.093,Z 436.331,A -85,B 0,C 180,E1 -7363.631,E2 -7363.631} C_VEL
LIN {X 0,Y 476.972,Z 532.163,A -85,B 0,C 180,E1 -7365.303,E2 -7365.303} C_VEL
LIN {X 0,Y 476.712,Z 543.895,A -85,B 0,C 180,E1 -7365.649,E2 -7365.649} C_VEL
LIN {X 0,Y 476.346,Z 556.361,A -85,B 0,C 180,E1 -7366.183,E2 -7366.183} C_VEL
LIN {X 0,Y 475.947,Z 568.677,A -85,B 0,C 180,E1 -7366.889,E2 -7366.889} C_VEL
LIN {X 0,Y 475.522,Z 580.307,A -85,B 0,C 180,E1 -7367.753,E2 -7367.753} C_VEL
LIN {X 0,Y 475.077,Z 591.521,A -85,B 0,C 180,E1 -7368.804,E2 -7368.804} C_VEL
LIN {X 0,Y 474.679,Z 599.897,A -85,B 0,C 180,E1 -7369.766,E2 -7369.766} C_VEL
LIN {X 0,Y 474.369,Z 608.957,A -85,B 0,C 180,E1 -7371.051,E2 -7371.051} C_VEL
LIN {X 0,Y 474.09,Z 616.248,A -85,B 0,C 180,E1 -7372.333,E2 -7372.333} C_VEL
LIN {X 0,Y 473.899,Z 621.718,A -85,B 0,C 180,E1 -7373.529,E2 -7373.529} C_VEL
LIN {X 0,Y 473.84,Z 626.619,A -85,B 0,C 180,E1 -7374.894,E2 -7374.894} C_VEL
LIN {X 0,Y 473.745,Z 628.999,A -85,B 0,C 180,E1 -7375.746,E2 -7375.746} C_VEL
LIN {X 0,Y 473.799,Z 630.944,A -85,B 0,C 180,E1 -7376.599,E2 -7376.599} C_VEL
LIN {X 0,Y 473.725,Z 632.452,A -85,B 0,C 180,E1 -7377.449,E2 -7377.449} C_VEL
LIN {X 0,Y 473.696,Z 633.495,A -85,B 0,C 180,E1 -7378.3,E2 -7378.3} C_VEL
LIN {X 0,Y 473.689,Z 634.141,A -85,B 0,C 180,E1 -7379.15,E2 -7379.15} C_VEL
LIN {X 0,Y 473.67,Z 634.391,A -85,B 0,C 180,E1 -7380,E2 -7380} C_VEL
LIN {X 0,Y 473.689,Z 634.191,A -85,B 0,C 180,E1 -7380.85,E2 -7380.85} C_VEL
LIN {X 0,Y 473.696,Z 633.58,A -85,B 0,C 180,E1 -7381.7,E2 -7381.7} C_VEL
LIN {X 0,Y 473.724,Z 632.573,A -85,B 0,C 180,E1 -7382.551,E2 -7382.551} C_VEL
LIN {X 0,Y 473.799,Z 631.135,A -85,B 0,C 180,E1 -7383.402,E2 -7383.402} C_VEL
LIN {X 0,Y 473.771,Z 628.136,A -85,B 0,C 180,E1 -7384.68,E2 -7384.68} C_VEL
LIN {X 0,Y 473.87,Z 623.212,A -85,B 0,C 180,E1 -7386.184,E2 -7386.184} C_VEL
LIN {X 0,Y 474.088,Z 616.769,A -85,B 0,C 180,E1 -7387.667,E2 -7387.667} C_VEL
LIN {X 0,Y 474.34,Z 609.617,A -85,B 0,C 180,E1 -7388.95,E2 -7388.95} C_VEL
LIN {X 0,Y 474.646,Z 600.727,A -85,B 0,C 180,E1 -7390.235,E2 -7390.235} C_VEL
LIN {X 0,Y 475.115,Z 590.51,A -85,B 0,C 180,E1 -7391.411,E2 -7391.411} C_VEL
LIN {X 0,Y 475.529,Z 580.629,A -85,B 0,C 180,E1 -7392.334,E2 -7392.334} C_VEL
LIN {X 0,Y 475.93,Z 569.299,A -85,B 0,C 180,E1 -7393.188,E2 -7393.188} C_VEL
LIN {X 0,Y 476.401,Z 556.534,A -85,B 0,C 180,E1 -7393.925,E2 -7393.925} C_VEL
LIN {X 0,Y 476.747,Z 544.131,A -85,B 0,C 180,E1 -7394.459,E2 -7394.459} C_VEL
LIN {X 0,Y 477.053,Z 531.273,A -85,B 0,C 180,E1 -7394.831,E2 -7394.831} C_VEL
LIN {X 0,Y 477.893,Z 434.844,A -85,B 0,C 180,E1 -7396.448,E2 -7396.448} C_VEL
LIN {X 0,Y 475.843,Z 420.853,A -85,B 0,C 180,E1 -7396.783,E2 -7396.783} C_VEL
LIN {X 0,Y 476.553,Z 397.429,A -85,B 0,C 180,E1 -7400.053,E2 -7400.053} C_VEL
LIN {X 0,Y 477.368,Z 373.468,A -85,B 0,C 180,E1 -7403.422,E2 -7403.422} C_VEL
LIN {X 0,Y 477.912,Z 356.216,A -85,B 0,C 180,E1 -7405.86,E2 -7405.86} C_VEL
LIN {X 0,Y 476.307,Z 347.265,A -85,B 0,C 180,E1 -7407.22,E2 -7407.22} C_VEL
LIN {X 0,Y 474.718,Z 340.102,A -85,B 0,C 180,E1 -7408.368,E2 -7408.368} C_VEL
LIN {X 0,Y 474.604,Z 339.991,A -85,B 0,C 180,E1 -7411.217,E2 -7411.217} C_VEL
LIN {X 0,Y 474.637,Z 339.991,A -85,B 0,C 180,E1 -7414.241,E2 -7414.241} C_VEL
LIN {X 0,Y 474.595,Z 339.989,A -85,B 0,C 180,E1 -7417.384,E2 -7417.384} C_VEL
LIN {X 0,Y 474.622,Z 339.989,A -85,B 0,C 180,E1 -7420.657,E2 -7420.657} C_VEL
LIN {X 0,Y 474.6,Z 339.986,A -85,B 0,C 180,E1 -7423.48,E2 -7423.48} C_VEL
LIN {X 0,Y 474.606,Z 339.992,A -85,B 0,C 180,E1 -7426.519,E2 -7426.519} C_VEL
LIN {X 0,Y 474.622,Z 339.984,A -85,B 0,C 180,E1 -7429.342,E2 -7429.342} C_VEL
LIN {X 0,Y 474.591,Z 339.989,A -85,B 0,C 180,E1 -7432.199,E2 -7432.199} C_VEL
LIN {X 0,Y 473.929,Z 340.073,A -85,B 0,C 180,E1 -7432.907,E2 -7432.907} C_VEL
LIN {X 0,Y 471.096,Z 340.43,A -85,B 0,C 180,E1 -7434.057,E2 -7434.057} C_VEL
LIN {X 0,Y 468.701,Z 340.729,A -85,B 0,C 180,E1 -7434.985,E2 -7434.985} C_VEL
LIN {X 0,Y 467.674,Z 340.856,A -85,B 0,C 180,E1 -7435.701,E2 -7435.701} C_VEL
LIN {X 0,Y 467.591,Z 340.865,A -85,B 0,C 180,E1 -7435.943,E2 -7435.943} C_VEL
LIN {X 0,Y 467.575,Z 340.867,A -85,B 0,C 180,E1 -7439.266,E2 -7439.266} C_VEL
LIN {X 0,Y 467.65,Z 340.857,A -85,B 0,C 180,E1 -7442.458,E2 -7442.458} C_VEL
LIN {X 0,Y 467.673,Z 340.94,A -85,B 0,C 180,E1 -7443.684,E2 -7443.684} C_VEL
LIN {X 0,Y 469.912,Z 351.768,A -85,B 0,C 180,E1 -7445.828,E2 -7445.828} C_VEL
LIN {X 0,Y 470.51,Z 356.36,A -85,B 0,C 180,E1 -7446.681,E2 -7446.681} C_VEL
LIN {X 0,Y 469.693,Z 372.17,A -85,B 0,C 180,E1 -7449.4,E2 -7449.4} C_VEL
LIN {X 0,Y 471.314,Z 380.557,A -85,B 0,C 180,E1 -7449.641,E2 -7449.641} C_VEL
LIN {X 0,Y 473.517,Z 392.2,A -85,B 0,C 180,E1 -7449.924,E2 -7449.924} C_VEL
LIN {X 0,Y 472.323,Z 509.092,A -85,B 0,C 180,E1 -7451.735,E2 -7451.735} C_VEL
LIN {X 0,Y 471.913,Z 523.604,A -85,B 0,C 180,E1 -7452.129,E2 -7452.129} C_VEL
LIN {X 0,Y 471.473,Z 536.762,A -85,B 0,C 180,E1 -7452.654,E2 -7452.654} C_VEL
LIN {X 0,Y 470.913,Z 549.3,A -85,B 0,C 180,E1 -7453.314,E2 -7453.314} C_VEL
LIN {X 0,Y 470.247,Z 562.074,A -85,B 0,C 180,E1 -7454.171,E2 -7454.171} C_VEL
LIN {X 0,Y 469.532,Z 573.812,A -85,B 0,C 180,E1 -7455.147,E2 -7455.147} C_VEL
LIN {X 0,Y 468.815,Z 585.525,A -85,B 0,C 180,E1 -7456.342,E2 -7456.342} C_VEL
LIN {X 0,Y 468.248,Z 594.711,A -85,B 0,C 180,E1 -7457.476,E2 -7457.476} C_VEL
LIN {X 0,Y 467.834,Z 603.269,A -85,B 0,C 180,E1 -7458.737,E2 -7458.737} C_VEL
LIN {X 0,Y 467.386,Z 611.796,A -85,B 0,C 180,E1 -7460.26,E2 -7460.26} C_VEL
LIN {X 0,Y 467.042,Z 618.671,A -85,B 0,C 180,E1 -7461.78,E2 -7461.78} C_VEL
LIN {X 0,Y 466.835,Z 623.417,A -85,B 0,C 180,E1 -7463.082,E2 -7463.082} C_VEL
LIN {X 0,Y 466.767,Z 628.33,A -85,B 0,C 180,E1 -7464.816,E2 -7464.816} C_VEL
LIN {X 0,Y 466.682,Z 631.754,A -85,B 0,C 180,E1 -7466.545,E2 -7466.545} C_VEL
LIN {X 0,Y 466.603,Z 633.793,A -85,B 0,C 180,E1 -7468.273,E2 -7468.273} C_VEL
LIN {X 0,Y 466.569,Z 634.497,A -85,B 0,C 180,E1 -7469.999,E2 -7469.999} C_VEL
LIN {X 0,Y 466.601,Z 633.875,A -85,B 0,C 180,E1 -7471.725,E2 -7471.725} C_VEL
LIN {X 0,Y 466.681,Z 631.913,A -85,B 0,C 180,E1 -7473.452,E2 -7473.452} C_VEL
LIN {X 0,Y 466.766,Z 628.56,A -85,B 0,C 180,E1 -7475.182,E2 -7475.182} C_VEL
LIN {X 0,Y 466.832,Z 623.719,A -85,B 0,C 180,E1 -7476.916,E2 -7476.916} C_VEL
LIN {X 0,Y 467.101,Z 617.246,A -85,B 0,C 180,E1 -7478.652,E2 -7478.652} C_VEL
LIN {X 0,Y 467.434,Z 610.04,A -85,B 0,C 180,E1 -7480.174,E2 -7480.174} C_VEL
LIN {X 0,Y 467.978,Z 601.128,A -85,B 0,C 180,E1 -7481.696,E2 -7481.696} C_VEL
LIN {X 0,Y 468.503,Z 591.769,A -85,B 0,C 180,E1 -7483.003,E2 -7483.003} C_VEL
LIN {X 0,Y 469.117,Z 581.402,A -85,B 0,C 180,E1 -7484.199,E2 -7484.199} C_VEL
LIN {X 0,Y 469.738,Z 569.97,A -85,B 0,C 180,E1 -7485.288,E2 -7485.288} C_VEL
LIN {X 0,Y 470.486,Z 557.303,A -85,B 0,C 180,E1 -7486.264,E2 -7486.264} C_VEL
LIN {X 0,Y 471.188,Z 544.039,A -85,B 0,C 180,E1 -7487.072,E2 -7487.072} C_VEL
LIN {X 0,Y 471.703,Z 530.04,A -85,B 0,C 180,E1 -7487.726,E2 -7487.726} C_VEL
LIN {X 0,Y 472.152,Z 516.237,A -85,B 0,C 180,E1 -7488.186,E2 -7488.186} C_VEL
LIN {X 0,Y 472.42,Z 502.033,A -85,B 0,C 180,E1 -7488.484,E2 -7488.484} C_VEL
LIN {X 0,Y 473.495,Z 392.057,A -85,B 0,C 180,E1 -7490.171,E2 -7490.171} C_VEL
LIN {X 0,Y 469.745,Z 372.647,A -85,B 0,C 180,E1 -7490.663,E2 -7490.663} C_VEL
LIN {X 0,Y 469.701,Z 371.827,A -85,B 0,C 180,E1 -7490.734,E2 -7490.734} C_VEL
LIN {X 0,Y 470.521,Z 355.587,A -85,B 0,C 180,E1 -7493.549,E2 -7493.549} C_VEL
LIN {X 0,Y 468.848,Z 346.432,A -85,B 0,C 180,E1 -7495.289,E2 -7495.289} C_VEL
LIN {X 0,Y 467.705,Z 341.246,A -85,B 0,C 180,E1 -7496.312,E2 -7496.312} C_VEL
LIN {X 0,Y 467.649,Z 340.848,A -85,B 0,C 180,E1 -7496.556,E2 -7496.556} C_VEL
LIN {X 0,Y 467.584,Z 340.847,A -85,B 0,C 180,E1 -7499.734,E2 -7499.734} C_VEL
LIN {X 0,Y 467.58,Z 340.861,A -85,B 0,C 180,E1 -7502.757,E2 -7502.757} C_VEL
LIN {X 0,Y 467.553,Z 340.865,A -85,B 0,C 180,E1 -7505.888,E2 -7505.888} C_VEL
LIN {X 0,Y 467.614,Z 340.857,A -85,B 0,C 180,E1 -7509.14,E2 -7509.14} C_VEL
LIN {X 0,Y 467.613,Z 340.86,A -85,B 0,C 180,E1 -7512.57,E2 -7512.57} C_VEL
LIN {X 0,Y 467.568,Z 340.86,A -85,B 0,C 180,E1 -7516.175,E2 -7516.175} C_VEL
LIN {X 0,Y 467.583,Z 340.863,A -85,B 0,C 180,E1 -7518.72,E2 -7518.72} C_VEL
LIN {X 0,Y 467.57,Z 340.854,A -85,B 0,C 180,E1 -7521.405,E2 -7521.405} C_VEL
LIN {X 0,Y 467.555,Z 340.865,A -85,B 0,C 180,E1 -7524.259,E2 -7524.259} C_VEL
LIN {X 0,Y 467.573,Z 340.868,A -85,B 0,C 180,E1 -7527.32,E2 -7527.32} C_VEL
LIN {X 0,Y 467.569,Z 340.841,A -85,B 0,C 180,E1 -7530.665,E2 -7530.665} C_VEL
LIN {X 0,Y 467.618,Z 340.848,A -85,B 0,C 180,E1 -7533.2,E2 -7533.2} C_VEL
LIN {X 0,Y 467.566,Z 340.866,A -85,B 0,C 180,E1 -7536.056,E2 -7536.056} C_VEL
LIN {X 0,Y 467.614,Z 340.86,A -85,B 0,C 180,E1 -7539.777,E2 -7539.777} C_VEL
LIN {X 0,Y 467.599,Z 340.859,A -85,B 0,C 180,E1 -7542.506,E2 -7542.506} C_VEL
LIN {X 0,Y 467.599,Z 340.857,A -85,B 0,C 180,E1 -7545.196,E2 -7545.196} C_VEL
LIN {X 0,Y 467.673,Z 340.85,A -85,B 0,C 180,E1 -7547.855,E2 -7547.855} C_VEL
LIN {X 0,Y 467.673,Z 340.85,A -85,B 0,C 180,E1 -7551.357,E2 -7551.357} C_VEL
LIN {X 0,Y 467.738,Z 340.842,A -85,B 0,C 180,E1 -7553.962,E2 -7553.962} C_VEL
LIN {X 0,Y 467.851,Z 340.828,A -85,B 0,C 180,E1 -7557.417,E2 -7557.417} C_VEL
LIN {X 0,Y 467.872,Z 340.826,A -85,B 0,C 180,E1 -7560,E2 -7560} C_VEL
LIN {X 0,Y 467.851,Z 340.828,A -85,B 0,C 180,E1 -7562.583,E2 -7562.583} C_VEL
LIN {X 0,Y 467.738,Z 340.842,A -85,B 0,C 180,E1 -7566.037,E2 -7566.037} C_VEL
LIN {X 0,Y 467.672,Z 340.851,A -85,B 0,C 180,E1 -7568.643,E2 -7568.643} C_VEL
LIN {X 0,Y 467.672,Z 340.85,A -85,B 0,C 180,E1 -7572.145,E2 -7572.145} C_VEL
LIN {X 0,Y 467.638,Z 340.846,A -85,B 0,C 180,E1 -7575.886,E2 -7575.886} C_VEL
LIN {X 0,Y 467.614,Z 340.856,A -85,B 0,C 180,E1 -7579.308,E2 -7579.308} C_VEL
LIN {X 0,Y 467.532,Z 340.863,A -85,B 0,C 180,E1 -7582.074,E2 -7582.074} C_VEL
LIN {X 0,Y 467.603,Z 340.86,A -85,B 0,C 180,E1 -7584.887,E2 -7584.887} C_VEL
LIN {X 0,Y 467.617,Z 340.844,A -85,B 0,C 180,E1 -7587.769,E2 -7587.769} C_VEL
LIN {X 0,Y 467.559,Z 340.86,A -85,B 0,C 180,E1 -7591.046,E2 -7591.046} C_VEL
LIN {X 0,Y 467.581,Z 340.869,A -85,B 0,C 180,E1 -7594.244,E2 -7594.244} C_VEL
LIN {X 0,Y 467.542,Z 340.851,A -85,B 0,C 180,E1 -7597.188,E2 -7597.188} C_VEL
LIN {X 0,Y 467.588,Z 340.862,A -85,B 0,C 180,E1 -7600.263,E2 -7600.263} C_VEL
LIN {X 0,Y 467.611,Z 340.859,A -85,B 0,C 180,E1 -7602.572,E2 -7602.572} C_VEL
LIN {X 0,Y 467.567,Z 340.862,A -85,B 0,C 180,E1 -7606.177,E2 -7606.177} C_VEL
LIN {X 0,Y 467.583,Z 340.86,A -85,B 0,C 180,E1 -7608.723,E2 -7608.723} C_VEL
LIN {X 0,Y 467.572,Z 340.862,A -85,B 0,C 180,E1 -7611.408,E2 -7611.408} C_VEL
LIN {X 0,Y 467.558,Z 340.864,A -85,B 0,C 180,E1 -7614.261,E2 -7614.261} C_VEL
LIN {X 0,Y 467.578,Z 340.861,A -85,B 0,C 180,E1 -7617.322,E2 -7617.322} C_VEL
LIN {X 0,Y 467.574,Z 340.846,A -85,B 0,C 180,E1 -7620.667,E2 -7620.667} C_VEL
LIN {X 0,Y 467.65,Z 340.931,A -85,B 0,C 180,E1 -7623.625,E2 -7623.625} C_VEL
LIN {X 0,Y 469.047,Z 347.491,A -85,B 0,C 180,E1 -7624.959,E2 -7624.959} C_VEL
LIN {X 0,Y 470.487,Z 355.335,A -85,B 0,C 180,E1 -7626.449,E2 -7626.449} C_VEL
LIN {X 0,Y 469.708,Z 372.058,A -85,B 0,C 180,E1 -7629.343,E2 -7629.343} C_VEL
LIN {X 0,Y 470.615,Z 377.13,A -85,B 0,C 180,E1 -7629.507,E2 -7629.507} C_VEL
LIN {X 0,Y 473.457,Z 391.626,A -85,B 0,C 180,E1 -7629.865,E2 -7629.865} C_VEL
LIN {X 0,Y 472.327,Z 508.735,A -85,B 0,C 180,E1 -7631.681,E2 -7631.681} C_VEL
LIN {X 0,Y 471.939,Z 522.822,A -85,B 0,C 180,E1 -7632.055,E2 -7632.055} C_VEL
LIN {X 0,Y 471.525,Z 535.696,A -85,B 0,C 180,E1 -7632.557,E2 -7632.557} C_VEL
LIN {X 0,Y 470.98,Z 548.432,A -85,B 0,C 180,E1 -7633.215,E2 -7633.215} C_VEL
LIN {X 0,Y 470.319,Z 561.273,A -85,B 0,C 180,E1 -7634.064,E2 -7634.064} C_VEL
LIN {X 0,Y 469.581,Z 573.151,A -85,B 0,C 180,E1 -7635.04,E2 -7635.04} C_VEL
LIN {X 0,Y 468.94,Z 584,A -85,B 0,C 180,E1 -7636.127,E2 -7636.127} C_VEL
LIN {X 0,Y 468.34,Z 593.479,A -85,B 0,C 180,E1 -7637.266,E2 -7637.266} C_VEL
LIN {X 0,Y 467.906,Z 602.211,A -85,B 0,C 180,E1 -7638.522,E2 -7638.522} C_VEL
LIN {X 0,Y 467.401,Z 610.926,A -85,B 0,C 180,E1 -7640.044,E2 -7640.044} C_VEL
LIN {X 0,Y 467.104,Z 617.06,A -85,B 0,C 180,E1 -7641.348,E2 -7641.348} C_VEL
LIN {X 0,Y 466.833,Z 623.572,A -85,B 0,C 180,E1 -7643.084,E2 -7643.084} C_VEL
LIN {X 0,Y 466.764,Z 628.45,A -85,B 0,C 180,E1 -7644.818,E2 -7644.818} C_VEL
LIN {X 0,Y 466.681,Z 631.838,A -85,B 0,C 180,E1 -7646.548,E2 -7646.548} C_VEL
LIN {X 0,Y 466.601,Z 633.838,A -85,B 0,C 180,E1 -7648.275,E2 -7648.275} C_VEL
LIN {X 0,Y 466.568,Z 634.5,A -85,B 0,C 180,E1 -7650.001,E2 -7650.001} C_VEL
LIN {X 0,Y 466.601,Z 633.834,A -85,B 0,C 180,E1 -7651.727,E2 -7651.727} C_VEL
LIN {X 0,Y 466.681,Z 631.829,A -85,B 0,C 180,E1 -7653.455,E2 -7653.455} C_VEL
LIN {X 0,Y 466.765,Z 628.44,A -85,B 0,C 180,E1 -7655.184,E2 -7655.184} C_VEL
LIN {X 0,Y 466.833,Z 623.565,A -85,B 0,C 180,E1 -7656.918,E2 -7656.918} C_VEL
LIN {X 0,Y 467.107,Z 617.048,A -85,B 0,C 180,E1 -7658.654,E2 -7658.654} C_VEL
LIN {X 0,Y 467.452,Z 609.795,A -85,B 0,C 180,E1 -7660.176,E2 -7660.176} C_VEL
LIN {X 0,Y 468.002,Z 600.812,A -85,B 0,C 180,E1 -7661.698,E2 -7661.698} C_VEL
LIN {X 0,Y 468.493,Z 591.38,A -85,B 0,C 180,E1 -7663.005,E2 -7663.005} C_VEL
LIN {X 0,Y 469.117,Z 580.937,A -85,B 0,C 180,E1 -7664.202,E2 -7664.202} C_VEL
LIN {X 0,Y 469.79,Z 569.407,A -85,B 0,C 180,E1 -7665.289,E2 -7665.289} C_VEL
LIN {X 0,Y 470.542,Z 556.611,A -85,B 0,C 180,E1 -7666.264,E2 -7666.264} C_VEL
LIN {X 0,Y 471.075,Z 544.746,A -85,B 0,C 180,E1 -7666.991,E2 -7666.991} C_VEL
LIN {X 0,Y 471.658,Z 530.994,A -85,B 0,C 180,E1 -7667.641,E2 -7667.641} C_VEL
LIN {X 0,Y 472.106,Z 517.764,A -85,B 0,C 180,E1 -7668.095,E2 -7668.095} C_VEL
LIN {X 0,Y 472.385,Z 504.027,A -85,B 0,C 180,E1 -7668.403,E2 -7668.403} C_VEL
LIN {X 0,Y 473.477,Z 392.911,A -85,B 0,C 180,E1 -7670.112,E2 -7670.112} C_VEL
LIN {X 0,Y 471.581,Z 381.871,A -85,B 0,C 180,E1 -7670.372,E2 -7670.372} C_VEL
LIN {X 0,Y 469.699,Z 372.311,A -85,B 0,C 180,E1 -7670.634,E2 -7670.634} C_VEL
LIN {X 0,Y 470.493,Z 356.614,A -85,B 0,C 180,E1 -7673.32,E2 -7673.32} C_VEL
LIN {X 0,Y 469.938,Z 351.97,A -85,B 0,C 180,E1 -7674.18,E2 -7674.18} C_VEL
LIN {X 0,Y 467.667,Z 341.055,A -85,B 0,C 180,E1 -7676.317,E2 -7676.317} C_VEL
LIN {X 0,Y 467.581,Z 340.85,A -85,B 0,C 180,E1 -7678.75,E2 -7678.75} C_VEL
LIN {X 0,Y 467.587,Z 340.866,A -85,B 0,C 180,E1 -7681.741,E2 -7681.741} C_VEL
LIN {X 0,Y 467.573,Z 340.866,A -85,B 0,C 180,E1 -7684.833,E2 -7684.833} C_VEL
LIN {X 0,Y 467.57,Z 340.869,A -85,B 0,C 180,E1 -7688.045,E2 -7688.045} C_VEL
LIN {X 0,Y 467.582,Z 340.864,A -85,B 0,C 180,E1 -7691.277,E2 -7691.277} C_VEL
LIN {X 0,Y 467.554,Z 340.873,A -85,B 0,C 180,E1 -7693.821,E2 -7693.821} C_VEL
LIN {X 0,Y 467.559,Z 340.869,A -85,B 0,C 180,E1 -7696.256,E2 -7696.256} C_VEL
LIN {X 0,Y 467.583,Z 340.865,A -85,B 0,C 180,E1 -7698.724,E2 -7698.724} C_VEL
LIN {X 0,Y 467.569,Z 340.869,A -85,B 0,C 180,E1 -7701.956,E2 -7701.956} C_VEL
LIN {X 0,Y 467.569,Z 340.868,A -85,B 0,C 180,E1 -7705.168,E2 -7705.168} C_VEL
LIN {X 0,Y 467.587,Z 340.867,A -85,B 0,C 180,E1 -7708.26,E2 -7708.26} C_VEL
LIN {X 0,Y 467.644,Z 341.011,A -85,B 0,C 180,E1 -7711.684,E2 -7711.684} C_VEL
LIN {X 0,Y 470.124,Z 351.529,A -85,B 0,C 180,E1 -7713.354,E2 -7713.354} C_VEL
LIN {X 0,Y 470.931,Z 357.225,A -85,B 0,C 180,E1 -7714.191,E2 -7714.191} C_VEL
LIN {X 0,Y 470.299,Z 378.596,A -85,B 0,C 180,E1 -7717.137,E2 -7717.137} C_VEL
LIN {X 0,Y 469.594,Z 401.507,A -85,B 0,C 180,E1 -7720.298,E2 -7720.298} C_VEL
LIN {X 0,Y 469.096,Z 420.813,A -85,B 0,C 180,E1 -7722.951,E2 -7722.951} C_VEL
LIN {X 0,Y 471.343,Z 436.973,A -85,B 0,C 180,E1 -7723.374,E2 -7723.374} C_VEL
LIN {X 0,Y 470.118,Z 531.995,A -85,B 0,C 180,E1 -7725.084,E2 -7725.084} C_VEL
LIN {X 0,Y 469.833,Z 543.718,A -85,B 0,C 180,E1 -7725.434,E2 -7725.434} C_VEL
LIN {X 0,Y 469.431,Z 556.197,A -85,B 0,C 180,E1 -7725.975,E2 -7725.975} C_VEL
LIN {X 0,Y 469.014,Z 568.517,A -85,B 0,C 180,E1 -7726.691,E2 -7726.691} C_VEL
LIN {X 0,Y 468.564,Z 579.513,A -85,B 0,C 180,E1 -7727.511,E2 -7727.511} C_VEL
LIN {X 0,Y 468.13,Z 590.365,A -85,B 0,C 180,E1 -7728.526,E2 -7728.526} C_VEL
LIN {X 0,Y 467.655,Z 599.808,A -85,B 0,C 180,E1 -7729.611,E2 -7729.611} C_VEL
LIN {X 0,Y 467.308,Z 608.887,A -85,B 0,C 180,E1 -7730.914,E2 -7730.914} C_VEL
LIN {X 0,Y 467.036,Z 616.191,A -85,B 0,C 180,E1 -7732.216,E2 -7732.216} C_VEL
LIN {X 0,Y 466.83,Z 622.068,A -85,B 0,C 180,E1 -7733.525,E2 -7733.525} C_VEL
LIN {X 0,Y 466.775,Z 626.595,A -85,B 0,C 180,E1 -7734.817,E2 -7734.817} C_VEL
LIN {X 0,Y 466.657,Z 628.981,A -85,B 0,C 180,E1 -7735.682,E2 -7735.682} C_VEL
LIN {X 0,Y 466.694,Z 630.93,A -85,B 0,C 180,E1 -7736.547,E2 -7736.547} C_VEL
LIN {X 0,Y 466.647,Z 632.44,A -85,B 0,C 180,E1 -7737.41,E2 -7737.41} C_VEL
LIN {X 0,Y 466.605,Z 633.485,A -85,B 0,C 180,E1 -7738.274,E2 -7738.274} C_VEL
LIN {X 0,Y 466.591,Z 634.131,A -85,B 0,C 180,E1 -7739.137,E2 -7739.137} C_VEL
LIN {X 0,Y 466.571,Z 634.378,A -85,B 0,C 180,E1 -7740,E2 -7740} C_VEL
LIN {X 0,Y 466.59,Z 634.172,A -85,B 0,C 180,E1 -7740.863,E2 -7740.863} C_VEL
LIN {X 0,Y 466.605,Z 633.555,A -85,B 0,C 180,E1 -7741.726,E2 -7741.726} C_VEL
LIN {X 0,Y 466.647,Z 632.541,A -85,B 0,C 180,E1 -7742.59,E2 -7742.59} C_VEL
LIN {X 0,Y 466.693,Z 631.089,A -85,B 0,C 180,E1 -7743.453,E2 -7743.453} C_VEL
LIN {X 0,Y 466.698,Z 628.068,A -85,B 0,C 180,E1 -7744.751,E2 -7744.751} C_VEL
LIN {X 0,Y 466.792,Z 623.964,A -85,B 0,C 180,E1 -7746.05,E2 -7746.05} C_VEL
LIN {X 0,Y 466.991,Z 617.658,A -85,B 0,C 180,E1 -7747.567,E2 -7747.567} C_VEL
LIN {X 0,Y 467.272,Z 610.764,A -85,B 0,C 180,E1 -7748.868,E2 -7748.868} C_VEL
LIN {X 0,Y 467.57,Z 602.094,A -85,B 0,C 180,E1 -7750.173,E2 -7750.173} C_VEL
LIN {X 0,Y 468.048,Z 592.261,A -85,B 0,C 180,E1 -7751.366,E2 -7751.366} C_VEL
LIN {X 0,Y 468.507,Z 581.715,A -85,B 0,C 180,E1 -7752.391,E2 -7752.391} C_VEL
LIN {X 0,Y 468.919,Z 571.262,A -85,B 0,C 180,E1 -7753.213,E2 -7753.213} C_VEL
LIN {X 0,Y 469.27,Z 560.949,A -85,B 0,C 180,E1 -7753.864,E2 -7753.864} C_VEL
LIN {X 0,Y 469.686,Z 548.749,A -85,B 0,C 180,E1 -7754.46,E2 -7754.46} C_VEL
LIN {X 0,Y 470.06,Z 535.298,A -85,B 0,C 180,E1 -7754.918,E2 -7754.918} C_VEL
LIN {X 0,Y 470.234,Z 520.859,A -85,B 0,C 180,E1 -7755.218,E2 -7755.218} C_VEL
LIN {X 0,Y 471.043,Z 435.656,A -85,B 0,C 180,E1 -7756.666,E2 -7756.666} C_VEL
LIN {X 0,Y 468.9,Z 420.951,A -85,B 0,C 180,E1 -7757.015,E2 -7757.015} C_VEL
LIN {X 0,Y 469.593,Z 398.756,A -85,B 0,C 180,E1 -7760.134,E2 -7760.134} C_VEL
LIN {X 0,Y 470.393,Z 376.233,A -85,B 0,C 180,E1 -7763.324,E2 -7763.324} C_VEL
LIN {X 0,Y 471.023,Z 357.287,A -85,B 0,C 180,E1 -7766.029,E2 -7766.029} C_VEL
LIN {X 0,Y 468.566,Z 345.047,A -85,B 0,C 180,E1 -7767.927,E2 -7767.927} C_VEL
LIN {X 0,Y 467.648,Z 340.95,A -85,B 0,C 180,E1 -7768.622,E2 -7768.622} C_VEL
LIN {X 0,Y 467.588,Z 340.866,A -85,B 0,C 180,E1 -7771.74,E2 -7771.74} C_VEL
LIN {X 0,Y 467.57,Z 340.867,A -85,B 0,C 180,E1 -7774.832,E2 -7774.832} C_VEL
LIN {X 0,Y 467.57,Z 340.869,A -85,B 0,C 180,E1 -7778.044,E2 -7778.044} C_VEL
LIN {X 0,Y 467.583,Z 340.862,A -85,B 0,C 180,E1 -7781.276,E2 -7781.276} C_VEL
LIN {X 0,Y 467.554,Z 340.864,A -85,B 0,C 180,E1 -7783.82,E2 -7783.82} C_VEL
LIN {X 0,Y 467.559,Z 340.864,A -85,B 0,C 180,E1 -7786.255,E2 -7786.255} C_VEL
LIN {X 0,Y 467.583,Z 340.862,A -85,B 0,C 180,E1 -7788.723,E2 -7788.723} C_VEL
LIN {X 0,Y 467.571,Z 340.868,A -85,B 0,C 180,E1 -7791.955,E2 -7791.955} C_VEL
LIN {X 0,Y 467.573,Z 340.864,A -85,B 0,C 180,E1 -7795.167,E2 -7795.167} C_VEL
LIN {X 0,Y 467.591,Z 340.865,A -85,B 0,C 180,E1 -7795.943,E2 -7795.943} C_VEL
LIN {X 0,Y 466.916,Z 340.948,A -85,B 0,C 180,E1 -7796.662,E2 -7796.662} C_VEL
LIN {X 0,Y 464.033,Z 341.305,A -85,B 0,C 180,E1 -7797.828,E2 -7797.828} C_VEL
LIN {X 0,Y 461.609,Z 341.609,A -85,B 0,C 180,E1 -7798.768,E2 -7798.768} C_VEL
LIN {X 0,Y 460.588,Z 341.732,A -85,B 0,C 180,E1 -7799.495,E2 -7799.495} C_VEL
LIN {X 0,Y 460.515,Z 341.736,A -85,B 0,C 180,E1 -7799.742,E2 -7799.742} C_VEL
LIN {X 0,Y 460.589,Z 341.74,A -85,B 0,C 180,E1 -7802.756,E2 -7802.756} C_VEL
LIN {X 0,Y 460.636,Z 341.862,A -85,B 0,C 180,E1 -7803.433,E2 -7803.433} C_VEL
LIN {X 0,Y 463.116,Z 353.749,A -85,B 0,C 180,E1 -7805.811,E2 -7805.811} C_VEL
LIN {X 0,Y 463.611,Z 357.67,A -85,B 0,C 180,E1 -7806.55,E2 -7806.55} C_VEL
LIN {X 0,Y 462.821,Z 372.279,A -85,B 0,C 180,E1 -7809.089,E2 -7809.089} C_VEL
LIN {X 0,Y 466.845,Z 393.545,A -85,B 0,C 180,E1 -7809.645,E2 -7809.645} C_VEL
LIN {X 0,Y 465.59,Z 509.113,A -85,B 0,C 180,E1 -7811.461,E2 -7811.461} C_VEL
LIN {X 0,Y 465.151,Z 523.617,A -85,B 0,C 180,E1 -7811.86,E2 -7811.86} C_VEL
LIN {X 0,Y 464.712,Z 536.771,A -85,B 0,C 180,E1 -7812.393,E2 -7812.393} C_VEL
LIN {X 0,Y 464.085,Z 549.483,A -85,B 0,C 180,E1 -7813.072,E2 -7813.072} C_VEL
LIN {X 0,Y 463.413,Z 562.08,A -85,B 0,C 180,E1 -7813.931,E2 -7813.931} C_VEL
LIN {X 0,Y 462.621,Z 573.817,A -85,B 0,C 180,E1 -7814.92,E2 -7814.92} C_VEL
LIN {X 0,Y 461.896,Z 585.529,A -85,B 0,C 180,E1 -7816.133,E2 -7816.133} C_VEL
LIN {X 0,Y 461.243,Z 595.332,A -85,B 0,C 180,E1 -7817.368,E2 -7817.368} C_VEL
LIN {X 0,Y 460.759,Z 604.626,A -85,B 0,C 180,E1 -7818.785,E2 -7818.785} C_VEL
LIN {X 0,Y 460.298,Z 612.903,A -85,B 0,C 180,E1 -7820.33,E2 -7820.33} C_VEL
LIN {X 0,Y 459.977,Z 618.673,A -85,B 0,C 180,E1 -7821.653,E2 -7821.653} C_VEL
LIN {X 0,Y 459.745,Z 623.419,A -85,B 0,C 180,E1 -7822.974,E2 -7822.974} C_VEL
LIN {X 0,Y 459.679,Z 628.331,A -85,B 0,C 180,E1 -7824.736,E2 -7824.736} C_VEL
LIN {X 0,Y 459.577,Z 631.754,A -85,B 0,C 180,E1 -7826.492,E2 -7826.492} C_VEL
LIN {X 0,Y 459.516,Z 633.793,A -85,B 0,C 180,E1 -7828.246,E2 -7828.246} C_VEL
LIN {X 0,Y 459.473,Z 634.497,A -85,B 0,C 180,E1 -7829.999,E2 -7829.999} C_VEL
LIN {X 0,Y 459.514,Z 633.875,A -85,B 0,C 180,E1 -7831.752,E2 -7831.752} C_VEL
LIN {X 0,Y 459.576,Z 631.912,A -85,B 0,C 180,E1 -7833.506,E2 -7833.506} C_VEL
LIN {X 0,Y 459.677,Z 628.559,A -85,B 0,C 180,E1 -7835.262,E2 -7835.262} C_VEL
LIN {X 0,Y 459.742,Z 623.718,A -85,B 0,C 180,E1 -7837.023,E2 -7837.023} C_VEL
LIN {X 0,Y 460.06,Z 617.244,A -85,B 0,C 180,E1 -7838.786,E2 -7838.786} C_VEL
LIN {X 0,Y 460.385,Z 610.038,A -85,B 0,C 180,E1 -7840.332,E2 -7840.332} C_VEL
LIN {X 0,Y 460.998,Z 601.125,A -85,B 0,C 180,E1 -7841.876,E2 -7841.876} C_VEL
LIN {X 0,Y 461.543,Z 591.765,A -85,B 0,C 180,E1 -7843.202,E2 -7843.202} C_VEL
LIN {X 0,Y 462.202,Z 581.398,A -85,B 0,C 180,E1 -7844.416,E2 -7844.416} C_VEL
LIN {X 0,Y 462.89,Z 569.965,A -85,B 0,C 180,E1 -7845.52,E2 -7845.52} C_VEL
LIN {X 0,Y 463.661,Z 557.296,A -85,B 0,C 180,E1 -7846.51,E2 -7846.51} C_VEL
LIN {X 0,Y 464.367,Z 544.692,A -85,B 0,C 180,E1 -7847.293,E2 -7847.293} C_VEL
LIN {X 0,Y 464.893,Z 531.33,A -85,B 0,C 180,E1 -7847.938,E2 -7847.938} C_VEL
LIN {X 0,Y 465.37,Z 518.053,A -85,B 0,C 180,E1 -7848.403,E2 -7848.403} C_VEL
LIN {X 0,Y 465.695,Z 503.607,A -85,B 0,C 180,E1 -7848.732,E2 -7848.732} C_VEL
LIN {X 0,Y 466.76,Z 392.454,A -85,B 0,C 180,E1 -7850.469,E2 -7850.469} C_VEL
LIN {X 0,Y 462.856,Z 372.405,A -85,B 0,C 180,E1 -7850.995,E2 -7850.995} C_VEL
LIN {X 0,Y 463.023,Z 367.59,A -85,B 0,C 180,E1 -7851.788,E2 -7851.788} C_VEL
LIN {X 0,Y 463.634,Z 356.892,A -85,B 0,C 180,E1 -7853.683,E2 -7853.683} C_VEL
LIN {X 0,Y 461.307,Z 345.039,A -85,B 0,C 180,E1 -7855.99,E2 -7855.99} C_VEL
LIN {X 0,Y 460.606,Z 341.819,A -85,B 0,C 180,E1 -7856.688,E2 -7856.688} C_VEL
LIN {X 0,Y 460.544,Z 341.722,A -85,B 0,C 180,E1 -7859.561,E2 -7859.561} C_VEL
LIN {X 0,Y 460.527,Z 341.739,A -85,B 0,C 180,E1 -7862.929,E2 -7862.929} C_VEL
LIN {X 0,Y 460.496,Z 341.743,A -85,B 0,C 180,E1 -7866.014,E2 -7866.014} C_VEL
LIN {X 0,Y 460.564,Z 341.735,A -85,B 0,C 180,E1 -7868.9,E2 -7868.9} C_VEL
LIN {X 0,Y 460.542,Z 341.745,A -85,B 0,C 180,E1 -7872.177,E2 -7872.177} C_VEL
LIN {X 0,Y 460.516,Z 341.731,A -85,B 0,C 180,E1 -7875.411,E2 -7875.411} C_VEL
LIN {X 0,Y 460.539,Z 341.742,A -85,B 0,C 180,E1 -7878.394,E2 -7878.394} C_VEL
LIN {X 0,Y 460.539,Z 341.73,A -85,B 0,C 180,E1 -7881.268,E2 -7881.268} C_VEL
LIN {X 0,Y 460.505,Z 341.741,A -85,B 0,C 180,E1 -7884.554,E2 -7884.554} C_VEL
LIN {X 0,Y 460.524,Z 341.742,A -85,B 0,C 180,E1 -7887.715,E2 -7887.715} C_VEL
LIN {X 0,Y 460.538,Z 341.716,A -85,B 0,C 180,E1 -7890.769,E2 -7890.769} C_VEL
LIN {X 0,Y 460.562,Z 341.735,A -85,B 0,C 180,E1 -7893.734,E2 -7893.734} C_VEL
LIN {X 0,Y 460.537,Z 341.74,A -85,B 0,C 180,E1 -7896.623,E2 -7896.623} C_VEL
LIN {X 0,Y 460.544,Z 341.738,A -85,B 0,C 180,E1 -7899.452,E2 -7899.452} C_VEL
LIN {X 0,Y 460.549,Z 341.737,A -85,B 0,C 180,E1 -7902.23,E2 -7902.23} C_VEL
LIN {X 0,Y 460.557,Z 341.731,A -85,B 0,C 180,E1 -7904.964,E2 -7904.964} C_VEL
LIN {X 0,Y 460.619,Z 341.73,A -85,B 0,C 180,E1 -7907.666,E2 -7907.666} C_VEL
LIN {X 0,Y 460.62,Z 341.726,A -85,B 0,C 180,E1 -7911.224,E2 -7911.224} C_VEL
LIN {X 0,Y 460.703,Z 341.719,A -85,B 0,C 180,E1 -7913.87,E2 -7913.87} C_VEL
LIN {X 0,Y 460.816,Z 341.704,A -85,B 0,C 180,E1 -7917.378,E2 -7917.378} C_VEL
LIN {X 0,Y 460.843,Z 341.702,A -85,B 0,C 180,E1 -7920,E2 -7920} C_VEL
LIN {X 0,Y 460.816,Z 341.704,A -85,B 0,C 180,E1 -7922.622,E2 -7922.622} C_VEL
LIN {X 0,Y 460.703,Z 341.719,A -85,B 0,C 180,E1 -7926.13,E2 -7926.13} C_VEL
LIN {X 0,Y 460.62,Z 341.727,A -85,B 0,C 180,E1 -7928.776,E2 -7928.776} C_VEL
LIN {X 0,Y 460.623,Z 341.73,A -85,B 0,C 180,E1 -7932.457,E2 -7932.457} C_VEL
LIN {X 0,Y 460.589,Z 341.724,A -85,B 0,C 180,E1 -7935.998,E2 -7935.998} C_VEL
LIN {X 0,Y 460.56,Z 341.739,A -85,B 0,C 180,E1 -7938.902,E2 -7938.902} C_VEL
LIN {X 0,Y 460.508,Z 341.736,A -85,B 0,C 180,E1 -7941.486,E2 -7941.486} C_VEL
LIN {X 0,Y 460.537,Z 341.744,A -85,B 0,C 180,E1 -7944.333,E2 -7944.333} C_VEL
LIN {X 0,Y 460.573,Z 341.721,A -85,B 0,C 180,E1 -7947.244,E2 -7947.244} C_VEL
LIN {X 0,Y 460.501,Z 341.725,A -85,B 0,C 180,E1 -7950.241,E2 -7950.241} C_VEL
LIN {X 0,Y 460.52,Z 341.742,A -85,B 0,C 180,E1 -7953.326,E2 -7953.326} C_VEL
LIN {X 0,Y 460.47,Z 341.736,A -85,B 0,C 180,E1 -7956.53,E2 -7956.53} C_VEL
LIN {X 0,Y 460.568,Z 341.731,A -85,B 0,C 180,E1 -7959.859,E2 -7959.859} C_VEL
LIN {X 0,Y 460.535,Z 341.737,A -85,B 0,C 180,E1 -7962.905,E2 -7962.905} C_VEL
LIN {X 0,Y 460.517,Z 341.735,A -85,B 0,C 180,E1 -7965.83,E2 -7965.83} C_VEL
LIN {X 0,Y 460.537,Z 341.737,A -85,B 0,C 180,E1 -7968.991,E2 -7968.991} C_VEL
LIN {X 0,Y 460.541,Z 341.738,A -85,B 0,C 180,E1 -7971.27,E2 -7971.27} C_VEL
LIN {X 0,Y 460.509,Z 341.743,A -85,B 0,C 180,E1 -7974.556,E2 -7974.556} C_VEL
LIN {X 0,Y 460.528,Z 341.741,A -85,B 0,C 180,E1 -7977.717,E2 -7977.717} C_VEL
LIN {X 0,Y 460.543,Z 341.721,A -85,B 0,C 180,E1 -7980.771,E2 -7980.771} C_VEL
LIN {X 0,Y 460.632,Z 341.851,A -85,B 0,C 180,E1 -7983.374,E2 -7983.374} C_VEL
LIN {X 0,Y 463.147,Z 354.029,A -85,B 0,C 180,E1 -7985.815,E2 -7985.815} C_VEL
LIN {X 0,Y 463.635,Z 357.952,A -85,B 0,C 180,E1 -7986.554,E2 -7986.554} C_VEL
LIN {X 0,Y 462.83,Z 372.099,A -85,B 0,C 180,E1 -7989.026,E2 -7989.026} C_VEL
LIN {X 0,Y 463.893,Z 377.763,A -85,B 0,C 180,E1 -7989.206,E2 -7989.206} C_VEL
LIN {X 0,Y 466.81,Z 393.322,A -85,B 0,C 180,E1 -7989.593,E2 -7989.593} C_VEL
LIN {X 0,Y 465.574,Z 509.975,A -85,B 0,C 180,E1 -7991.434,E2 -7991.434} C_VEL
LIN {X 0,Y 465.132,Z 524.439,A -85,B 0,C 180,E1 -7991.844,E2 -7991.844} C_VEL
LIN {X 0,Y 464.687,Z 537.738,A -85,B 0,C 180,E1 -7992.395,E2 -7992.395} C_VEL
LIN {X 0,Y 464.044,Z 550.267,A -85,B 0,C 180,E1 -7993.074,E2 -7993.074} C_VEL
LIN {X 0,Y 463.392,Z 562.701,A -85,B 0,C 180,E1 -7993.933,E2 -7993.933} C_VEL
LIN {X 0,Y 462.62,Z 574.326,A -85,B 0,C 180,E1 -7994.922,E2 -7994.922} C_VEL
LIN {X 0,Y 461.872,Z 585.952,A -85,B 0,C 180,E1 -7996.135,E2 -7996.135} C_VEL
LIN {X 0,Y 461.239,Z 595.685,A -85,B 0,C 180,E1 -7997.37,E2 -7997.37} C_VEL
LIN {X 0,Y 460.75,Z 604.92,A -85,B 0,C 180,E1 -7998.787,E2 -7998.787} C_VEL
LIN {X 0,Y 460.285,Z 613.128,A -85,B 0,C 180,E1 -8000.332,E2 -8000.332} C_VEL
LIN {X 0,Y 459.967,Z 618.868,A -85,B 0,C 180,E1 -8001.655,E2 -8001.655} C_VEL
LIN {X 0,Y 459.743,Z 623.572,A -85,B 0,C 180,E1 -8002.977,E2 -8002.977} C_VEL
LIN {X 0,Y 459.676,Z 628.45,A -85,B 0,C 180,E1 -8004.738,E2 -8004.738} C_VEL
LIN {X 0,Y 459.576,Z 631.838,A -85,B 0,C 180,E1 -8006.494,E2 -8006.494} C_VEL
LIN {X 0,Y 459.513,Z 633.838,A -85,B 0,C 180,E1 -8008.248,E2 -8008.248} C_VEL
LIN {X 0,Y 459.472,Z 634.5,A -85,B 0,C 180,E1 -8010.001,E2 -8010.001} C_VEL
LIN {X 0,Y 459.514,Z 633.834,A -85,B 0,C 180,E1 -8011.754,E2 -8011.754} C_VEL
LIN {X 0,Y 459.577,Z 631.829,A -85,B 0,C 180,E1 -8013.508,E2 -8013.508} C_VEL
LIN {X 0,Y 459.677,Z 628.44,A -85,B 0,C 180,E1 -8015.264,E2 -8015.264} C_VEL
LIN {X 0,Y 459.743,Z 623.564,A -85,B 0,C 180,E1 -8017.026,E2 -8017.026} C_VEL
LIN {X 0,Y 460.064,Z 617.047,A -85,B 0,C 180,E1 -8018.788,E2 -8018.788} C_VEL
LIN {X 0,Y 460.409,Z 609.794,A -85,B 0,C 180,E1 -8020.334,E2 -8020.334} C_VEL
LIN {X 0,Y 461.027,Z 600.811,A -85,B 0,C 180,E1 -8021.877,E2 -8021.877} C_VEL
LIN {X 0,Y 461.54,Z 591.378,A -85,B 0,C 180,E1 -8023.204,E2 -8023.204} C_VEL
LIN {X 0,Y 462.213,Z 580.935,A -85,B 0,C 180,E1 -8024.418,E2 -8024.418} C_VEL
LIN {X 0,Y 462.908,Z 569.404,A -85,B 0,C 180,E1 -8025.522,E2 -8025.522} C_VEL
LIN {X 0,Y 463.706,Z 556.607,A -85,B 0,C 180,E1 -8026.511,E2 -8026.511} C_VEL
LIN {X 0,Y 464.36,Z 543.538,A -85,B 0,C 180,E1 -8027.313,E2 -8027.313} C_VEL
LIN {X 0,Y 464.938,Z 529.817,A -85,B 0,C 180,E1 -8027.956,E2 -8027.956} C_VEL
LIN {X 0,Y 465.411,Z 516.749,A -85,B 0,C 180,E1 -8028.395,E2 -8028.395} C_VEL
LIN {X 0,Y 465.689,Z 502.483,A -85,B 0,C 180,E1 -8028.706,E2 -8028.706} C_VEL
LIN {X 0,Y 466.828,Z 393.374,A -85,B 0,C 180,E1 -8030.403,E2 -8030.403} C_VEL
LIN {X 0,Y 462.829,Z 372.268,A -85,B 0,C 180,E1 -8030.957,E2 -8030.957} C_VEL
LIN {X 0,Y 463.61,Z 357.92,A -85,B 0,C 180,E1 -8033.45,E2 -8033.45} C_VEL
LIN {X 0,Y 462.653,Z 351.318,A -85,B 0,C 180,E1 -8034.705,E2 -8034.705} C_VEL
LIN {X 0,Y 460.632,Z 341.826,A -85,B 0,C 180,E1 -8036.628,E2 -8036.628} C_VEL
LIN {X 0,Y 460.535,Z 341.732,A -85,B 0,C 180,E1 -8039.559,E2 -8039.559} C_VEL
LIN {X 0,Y 460.536,Z 341.746,A -85,B 0,C 180,E1 -8042.285,E2 -8042.285} C_VEL
LIN {X 0,Y 460.519,Z 341.746,A -85,B 0,C 180,E1 -8045.446,E2 -8045.446} C_VEL
LIN {X 0,Y 460.549,Z 341.741,A -85,B 0,C 180,E1 -8048.898,E2 -8048.898} C_VEL
LIN {X 0,Y 460.527,Z 341.746,A -85,B 0,C 180,E1 -8052.182,E2 -8052.182} C_VEL
LIN {X 0,Y 460.518,Z 341.746,A -85,B 0,C 180,E1 -8055.412,E2 -8055.412} C_VEL
LIN {X 0,Y 460.537,Z 341.744,A -85,B 0,C 180,E1 -8058.398,E2 -8058.398} C_VEL
LIN {X 0,Y 460.531,Z 341.744,A -85,B 0,C 180,E1 -8061.267,E2 -8061.267} C_VEL
LIN {X 0,Y 460.515,Z 341.746,A -85,B 0,C 180,E1 -8064.555,E2 -8064.555} C_VEL
LIN {X 0,Y 460.536,Z 341.746,A -85,B 0,C 180,E1 -8067.716,E2 -8067.716} C_VEL
LIN {X 0,Y 460.57,Z 341.873,A -85,B 0,C 180,E1 -8071.318,E2 -8071.318} C_VEL
LIN {X 0,Y 462.985,Z 351.604,A -85,B 0,C 180,E1 -8072.91,E2 -8072.91} C_VEL
LIN {X 0,Y 464.185,Z 358.463,A -85,B 0,C 180,E1 -8073.955,E2 -8073.955} C_VEL
LIN {X 0,Y 463.533,Z 378.667,A -85,B 0,C 180,E1 -8076.784,E2 -8076.784} C_VEL
LIN {X 0,Y 462.86,Z 398.596,A -85,B 0,C 180,E1 -8079.56,E2 -8079.56} C_VEL
LIN {X 0,Y 462.222,Z 420.651,A -85,B 0,C 180,E1 -8082.63,E2 -8082.63} C_VEL
LIN {X 0,Y 464.607,Z 436.878,A -85,B 0,C 180,E1 -8083.088,E2 -8083.088} C_VEL
LIN {X 0,Y 463.417,Z 521.235,A -85,B 0,C 180,E1 -8084.638,E2 -8084.638} C_VEL
LIN {X 0,Y 463.16,Z 536.151,A -85,B 0,C 180,E1 -8084.967,E2 -8084.967} C_VEL
LIN {X 0,Y 462.811,Z 549.213,A -85,B 0,C 180,E1 -8085.433,E2 -8085.433} C_VEL
LIN {X 0,Y 462.389,Z 561.207,A -85,B 0,C 180,E1 -8086.037,E2 -8086.037} C_VEL
LIN {X 0,Y 461.891,Z 573.67,A -85,B 0,C 180,E1 -8086.859,E2 -8086.859} C_VEL
LIN {X 0,Y 461.41,Z 584.798,A -85,B 0,C 180,E1 -8087.799,E2 -8087.799} C_VEL
LIN {X 0,Y 460.92,Z 594.316,A -85,B 0,C 180,E1 -8088.79,E2 -8088.79} C_VEL
LIN {X 0,Y 460.571,Z 603.018,A -85,B 0,C 180,E1 -8089.893,E2 -8089.893} C_VEL
LIN {X 0,Y 460.18,Z 611.475,A -85,B 0,C 180,E1 -8091.215,E2 -8091.215} C_VEL
LIN {X 0,Y 459.88,Z 618.255,A -85,B 0,C 180,E1 -8092.536,E2 -8092.536} C_VEL
LIN {X 0,Y 459.722,Z 623.656,A -85,B 0,C 180,E1 -8093.857,E2 -8093.857} C_VEL
LIN {X 0,Y 459.63,Z 627.839,A -85,B 0,C 180,E1 -8095.176,E2 -8095.176} C_VEL
LIN {X 0,Y 459.59,Z 630.926,A -85,B 0,C 180,E1 -8096.493,E2 -8096.493} C_VEL
LIN {X 0,Y 459.571,Z 632.435,A -85,B 0,C 180,E1 -8097.371,E2 -8097.371} C_VEL
LIN {X 0,Y 459.518,Z 633.479,A -85,B 0,C 180,E1 -8098.247,E2 -8098.247} C_VEL
LIN {X 0,Y 459.496,Z 634.123,A -85,B 0,C 180,E1 -8099.124,E2 -8099.124} C_VEL
LIN {X 0,Y 459.475,Z 634.365,A -85,B 0,C 180,E1 -8100,E2 -8100} C_VEL
LIN {X 0,Y 459.496,Z 634.15,A -85,B 0,C 180,E1 -8100.876,E2 -8100.876} C_VEL
LIN {X 0,Y 459.518,Z 633.525,A -85,B 0,C 180,E1 -8101.753,E2 -8101.753} C_VEL
LIN {X 0,Y 459.571,Z 632.501,A -85,B 0,C 180,E1 -8102.63,E2 -8102.63} C_VEL
LIN {X 0,Y 459.589,Z 631.03,A -85,B 0,C 180,E1 -8103.507,E2 -8103.507} C_VEL
LIN {X 0,Y 459.629,Z 627.983,A -85,B 0,C 180,E1 -8104.824,E2 -8104.824} C_VEL
LIN {X 0,Y 459.716,Z 623.848,A -85,B 0,C 180,E1 -8106.143,E2 -8106.143} C_VEL
LIN {X 0,Y 459.923,Z 617.499,A -85,B 0,C 180,E1 -8107.684,E2 -8107.684} C_VEL
LIN {X 0,Y 460.192,Z 610.551,A -85,B 0,C 180,E1 -8109.006,E2 -8109.006} C_VEL
LIN {X 0,Y 460.524,Z 601.82,A -85,B 0,C 180,E1 -8110.33,E2 -8110.33} C_VEL
LIN {X 0,Y 461.027,Z 591.909,A -85,B 0,C 180,E1 -8111.542,E2 -8111.542} C_VEL
LIN {X 0,Y 461.497,Z 582.53,A -85,B 0,C 180,E1 -8112.47,E2 -8112.47} C_VEL
LIN {X 0,Y 461.955,Z 570.718,A -85,B 0,C 180,E1 -8113.415,E2 -8113.415} C_VEL
LIN {X 0,Y 462.388,Z 559.296,A -85,B 0,C 180,E1 -8114.131,E2 -8114.131} C_VEL
LIN {X 0,Y 462.838,Z 546.415,A -85,B 0,C 180,E1 -8114.735,E2 -8114.735} C_VEL
LIN {X 0,Y 463.16,Z 533.991,A -85,B 0,C 180,E1 -8115.146,E2 -8115.146} C_VEL
LIN {X 0,Y 463.389,Z 515.567,A -85,B 0,C 180,E1 -8115.504,E2 -8115.504} C_VEL
LIN {X 0,Y 464.266,Z 436.806,A -85,B 0,C 180,E1 -8116.873,E2 -8116.873} C_VEL
LIN {X 0,Y 461.983,Z 421.044,A -85,B 0,C 180,E1 -8117.255,E2 -8117.255} C_VEL
LIN {X 0,Y 462.712,Z 398.418,A -85,B 0,C 180,E1 -8120.447,E2 -8120.447} C_VEL
LIN {X 0,Y 463.551,Z 375.783,A -85,B 0,C 180,E1 -8123.689,E2 -8123.689} C_VEL
LIN {X 0,Y 464.142,Z 359.418,A -85,B 0,C 180,E1 -8126.048,E2 -8126.048} C_VEL
LIN {X 0,Y 463.011,Z 352.648,A -85,B 0,C 180,E1 -8127.089,E2 -8127.089} C_VEL
LIN {X 0,Y 460.585,Z 341.838,A -85,B 0,C 180,E1 -8128.853,E2 -8128.853} C_VEL
LIN {X 0,Y 460.537,Z 341.747,A -85,B 0,C 180,E1 -8132.284,E2 -8132.284} C_VEL
LIN {X 0,Y 460.516,Z 341.744,A -85,B 0,C 180,E1 -8135.445,E2 -8135.445} C_VEL
LIN {X 0,Y 460.539,Z 341.741,A -85,B 0,C 180,E1 -8138.896,E2 -8138.896} C_VEL
LIN {X 0,Y 460.528,Z 341.747,A -85,B 0,C 180,E1 -8142.181,E2 -8142.181} C_VEL
LIN {X 0,Y 460.519,Z 341.73,A -85,B 0,C 180,E1 -8145.411,E2 -8145.411} C_VEL
LIN {X 0,Y 460.537,Z 341.742,A -85,B 0,C 180,E1 -8148.397,E2 -8148.397} C_VEL
LIN {X 0,Y 460.532,Z 341.738,A -85,B 0,C 180,E1 -8151.267,E2 -8151.267} C_VEL
LIN {X 0,Y 460.518,Z 341.742,A -85,B 0,C 180,E1 -8154.554,E2 -8154.554} C_VEL
LIN {X 0,Y 460.537,Z 341.74,A -85,B 0,C 180,E1 -8157.715,E2 -8157.715} C_VEL
LIN {X 0,Y 460.515,Z 341.736,A -85,B 0,C 180,E1 -8159.742,E2 -8159.742} C_VEL
LIN {X 0,Y 459.86,Z 341.816,A -85,B 0,C 180,E1 -8160.229,E2 -8160.229} C_VEL
LIN {X 0,Y 457.04,Z 342.163,A -85,B 0,C 180,E1 -8160.993,E2 -8160.993} C_VEL
LIN {X 0,Y 454.205,Z 342.517,A -85,B 0,C 180,E1 -8161.765,E2 -8161.765} C_VEL
LIN {X 0,Y 453.547,Z 342.607,A -85,B 0,C 180,E1 -8162.263,E2 -8162.263} C_VEL
LIN {X 0,Y 453.59,Z 342.791,A -85,B 0,C 180,E1 -8163.174,E2 -8163.174} C_VEL
LIN {X 0,Y 456.105,Z 354.731,A -85,B 0,C 180,E1 -8165.596,E2 -8165.596} C_VEL
LIN {X 0,Y 456.711,Z 358.98,A -85,B 0,C 180,E1 -8166.415,E2 -8166.415} C_VEL
LIN {X 0,Y 455.974,Z 372.042,A -85,B 0,C 180,E1 -8168.734,E2 -8168.734} C_VEL
LIN {X 0,Y 456.498,Z 375.079,A -85,B 0,C 180,E1 -8168.857,E2 -8168.857} C_VEL
LIN {X 0,Y 460.182,Z 394.11,A -85,B 0,C 180,E1 -8169.346,E2 -8169.346} C_VEL
LIN {X 0,Y 458.873,Z 509.134,A -85,B 0,C 180,E1 -8171.179,E2 -8171.179} C_VEL
LIN {X 0,Y 458.403,Z 523.21,A -85,B 0,C 180,E1 -8171.568,E2 -8171.568} C_VEL
LIN {X 0,Y 457.934,Z 536.78,A -85,B 0,C 180,E1 -8172.124,E2 -8172.124} C_VEL
LIN {X 0,Y 457.277,Z 549.668,A -85,B 0,C 180,E1 -8172.824,E2 -8172.824} C_VEL
LIN {X 0,Y 456.591,Z 562.085,A -85,B 0,C 180,E1 -8173.684,E2 -8173.684} C_VEL
LIN {X 0,Y 455.764,Z 573.822,A -85,B 0,C 180,E1 -8174.687,E2 -8174.687} C_VEL
LIN {X 0,Y 454.977,Z 585.533,A -85,B 0,C 180,E1 -8175.918,E2 -8175.918} C_VEL
LIN {X 0,Y 454.245,Z 595.935,A -85,B 0,C 180,E1 -8177.254,E2 -8177.254} C_VEL
LIN {X 0,Y 453.768,Z 604.628,A -85,B 0,C 180,E1 -8178.61,E2 -8178.61} C_VEL
LIN {X 0,Y 453.268,Z 612.905,A -85,B 0,C 180,E1 -8180.179,E2 -8180.179} C_VEL
LIN {X 0,Y 452.932,Z 618.674,A -85,B 0,C 180,E1 -8181.522,E2 -8181.522} C_VEL
LIN {X 0,Y 452.672,Z 623.42,A -85,B 0,C 180,E1 -8182.864,E2 -8182.864} C_VEL
LIN {X 0,Y 452.595,Z 628.332,A -85,B 0,C 180,E1 -8184.653,E2 -8184.653} C_VEL
LIN {X 0,Y 452.475,Z 631.755,A -85,B 0,C 180,E1 -8186.437,E2 -8186.437} C_VEL
LIN {X 0,Y 452.432,Z 633.794,A -85,B 0,C 180,E1 -8188.219,E2 -8188.219} C_VEL
LIN {X 0,Y 452.38,Z 634.497,A -85,B 0,C 180,E1 -8189.999,E2 -8189.999} C_VEL
LIN {X 0,Y 452.43,Z 633.874,A -85,B 0,C 180,E1 -8191.779,E2 -8191.779} C_VEL
LIN {X 0,Y 452.473,Z 631.912,A -85,B 0,C 180,E1 -8193.561,E2 -8193.561} C_VEL
LIN {X 0,Y 452.594,Z 628.558,A -85,B 0,C 180,E1 -8195.345,E2 -8195.345} C_VEL
LIN {X 0,Y 452.668,Z 623.716,A -85,B 0,C 180,E1 -8197.134,E2 -8197.134} C_VEL
LIN {X 0,Y 453.001,Z 617.242,A -85,B 0,C 180,E1 -8198.924,E2 -8198.924} C_VEL
LIN {X 0,Y 453.362,Z 610.035,A -85,B 0,C 180,E1 -8200.494,E2 -8200.494} C_VEL
LIN {X 0,Y 454.02,Z 601.122,A -85,B 0,C 180,E1 -8202.061,E2 -8202.061} C_VEL
LIN {X 0,Y 454.591,Z 591.761,A -85,B 0,C 180,E1 -8203.408,E2 -8203.408} C_VEL
LIN {X 0,Y 455.277,Z 581.393,A -85,B 0,C 180,E1 -8204.641,E2 -8204.641} C_VEL
LIN {X 0,Y 456.052,Z 569.96,A -85,B 0,C 180,E1 -8205.759,E2 -8205.759} C_VEL
LIN {X 0,Y 456.82,Z 557.29,A -85,B 0,C 180,E1 -8206.765,E2 -8206.765} C_VEL
LIN {X 0,Y 457.608,Z 544.113,A -85,B 0,C 180,E1 -8207.59,E2 -8207.59} C_VEL
LIN {X 0,Y 458.154,Z 531.309,A -85,B 0,C 180,E1 -8208.212,E2 -8208.212} C_VEL
LIN {X 0,Y 458.643,Z 518.036,A -85,B 0,C 180,E1 -8208.683,E2 -8208.683} C_VEL
LIN {X 0,Y 458.981,Z 503.583,A -85,B 0,C 180,E1 -8209.016,E2 -8209.016} C_VEL
LIN {X 0,Y 460.131,Z 393.672,A -85,B 0,C 180,E1 -8210.757,E2 -8210.757} C_VEL
LIN {X 0,Y 455.998,Z 372.315,A -85,B 0,C 180,E1 -8211.33,E2 -8211.33} C_VEL
LIN {X 0,Y 456.739,Z 358.198,A -85,B 0,C 180,E1 -8213.822,E2 -8213.822} C_VEL
LIN {X 0,Y 454.196,Z 345.573,A -85,B 0,C 180,E1 -8216.327,E2 -8216.327} C_VEL
LIN {X 0,Y 453.569,Z 342.672,A -85,B 0,C 180,E1 -8216.98,E2 -8216.98} C_VEL
LIN {X 0,Y 453.486,Z 342.602,A -85,B 0,C 180,E1 -8219.787,E2 -8219.787} C_VEL
LIN {X 0,Y 453.487,Z 342.616,A -85,B 0,C 180,E1 -8223.188,E2 -8223.188} C_VEL
LIN {X 0,Y 453.452,Z 342.622,A -85,B 0,C 180,E1 -8226.298,E2 -8226.298} C_VEL
LIN {X 0,Y 453.528,Z 342.61,A -85,B 0,C 180,E1 -8229.444,E2 -8229.444} C_VEL
LIN {X 0,Y 453.486,Z 342.619,A -85,B 0,C 180,E1 -8232.99,E2 -8232.99} C_VEL
LIN {X 0,Y 453.47,Z 342.61,A -85,B 0,C 180,E1 -8235.779,E2 -8235.779} C_VEL
LIN {X 0,Y 453.49,Z 342.621,A -85,B 0,C 180,E1 -8238.21,E2 -8238.21} C_VEL
LIN {X 0,Y 453.525,Z 342.605,A -85,B 0,C 180,E1 -8240.786,E2 -8240.786} C_VEL
LIN {X 0,Y 453.449,Z 342.617,A -85,B 0,C 180,E1 -8243.916,E2 -8243.916} C_VEL
LIN {X 0,Y 453.475,Z 342.623,A -85,B 0,C 180,E1 -8247.15,E2 -8247.15} C_VEL
LIN {X 0,Y 453.505,Z 342.592,A -85,B 0,C 180,E1 -8250.27,E2 -8250.27} C_VEL
LIN {X 0,Y 453.506,Z 342.606,A -85,B 0,C 180,E1 -8253.294,E2 -8253.294} C_VEL
LIN {X 0,Y 453.495,Z 342.618,A -85,B 0,C 180,E1 -8256.238,E2 -8256.238} C_VEL
LIN {X 0,Y 453.483,Z 342.614,A -85,B 0,C 180,E1 -8259.118,E2 -8259.118} C_VEL
LIN {X 0,Y 453.502,Z 342.616,A -85,B 0,C 180,E1 -8261.944,E2 -8261.944} C_VEL
LIN {X 0,Y 453.53,Z 342.604,A -85,B 0,C 180,E1 -8264.726,E2 -8264.726} C_VEL
LIN {X 0,Y 453.591,Z 342.608,A -85,B 0,C 180,E1 -8267.472,E2 -8267.472} C_VEL
LIN {X 0,Y 453.584,Z 342.601,A -85,B 0,C 180,E1 -8271.086,E2 -8271.086} C_VEL
LIN {X 0,Y 453.67,Z 342.595,A -85,B 0,C 180,E1 -8273.775,E2 -8273.775} C_VEL
LIN {X 0,Y 453.757,Z 342.582,A -85,B 0,C 180,E1 -8277.337,E2 -8277.337} C_VEL
LIN {X 0,Y 453.814,Z 342.577,A -85,B 0,C 180,E1 -8280,E2 -8280} C_VEL
LIN {X 0,Y 453.757,Z 342.583,A -85,B 0,C 180,E1 -8282.663,E2 -8282.663} C_VEL
LIN {X 0,Y 453.67,Z 342.595,A -85,B 0,C 180,E1 -8286.225,E2 -8286.225} C_VEL
LIN {X 0,Y 453.583,Z 342.601,A -85,B 0,C 180,E1 -8288.913,E2 -8288.913} C_VEL
LIN {X 0,Y 453.59,Z 342.607,A -85,B 0,C 180,E1 -8292.551,E2 -8292.551} C_VEL
LIN {X 0,Y 453.533,Z 342.603,A -85,B 0,C 180,E1 -8296.196,E2 -8296.196} C_VEL
LIN {X 0,Y 453.51,Z 342.615,A -85,B 0,C 180,E1 -8299.041,E2 -8299.041} C_VEL
LIN {X 0,Y 453.468,Z 342.613,A -85,B 0,C 180,E1 -8301.836,E2 -8301.836} C_VEL
LIN {X 0,Y 453.515,Z 342.617,A -85,B 0,C 180,E1 -8304.734,E2 -8304.734} C_VEL
LIN {X 0,Y 453.527,Z 342.596,A -85,B 0,C 180,E1 -8307.962,E2 -8307.962} C_VEL
LIN {X 0,Y 453.457,Z 342.615,A -85,B 0,C 180,E1 -8311.526,E2 -8311.526} C_VEL
LIN {X 0,Y 453.48,Z 342.619,A -85,B 0,C 180,E1 -8314.779,E2 -8314.779} C_VEL
LIN {X 0,Y 453.475,Z 342.603,A -85,B 0,C 180,E1 -8318.311,E2 -8318.311} C_VEL
LIN {X 0,Y 453.508,Z 342.619,A -85,B 0,C 180,E1 -8320.607,E2 -8320.607} C_VEL
LIN {X 0,Y 453.474,Z 342.616,A -85,B 0,C 180,E1 -8323.249,E2 -8323.249} C_VEL
LIN {X 0,Y 453.47,Z 342.611,A -85,B 0,C 180,E1 -8325.782,E2 -8325.782} C_VEL
LIN {X 0,Y 453.49,Z 342.621,A -85,B 0,C 180,E1 -8328.212,E2 -8328.212} C_VEL
LIN {X 0,Y 453.526,Z 342.612,A -85,B 0,C 180,E1 -8330.788,E2 -8330.788} C_VEL
LIN {X 0,Y 453.452,Z 342.621,A -85,B 0,C 180,E1 -8333.919,E2 -8333.919} C_VEL
LIN {X 0,Y 453.479,Z 342.617,A -85,B 0,C 180,E1 -8337.153,E2 -8337.153} C_VEL
LIN {X 0,Y 453.51,Z 342.599,A -85,B 0,C 180,E1 -8340.272,E2 -8340.272} C_VEL
LIN {X 0,Y 453.582,Z 342.774,A -85,B 0,C 180,E1 -8343.114,E2 -8343.114} C_VEL
LIN {X 0,Y 456.147,Z 354.919,A -85,B 0,C 180,E1 -8345.584,E2 -8345.584} C_VEL
LIN {X 0,Y 456.748,Z 359.261,A -85,B 0,C 180,E1 -8346.419,E2 -8346.419} C_VEL
LIN {X 0,Y 455.983,Z 372.153,A -85,B 0,C 180,E1 -8348.701,E2 -8348.701} C_VEL
LIN {X 0,Y 457.798,Z 381.419,A -85,B 0,C 180,E1 -8348.976,E2 -8348.976} C_VEL
LIN {X 0,Y 460.19,Z 394.765,A -85,B 0,C 180,E1 -8349.309,E2 -8349.309} C_VEL
LIN {X 0,Y 458.871,Z 508.761,A -85,B 0,C 180,E1 -8351.124,E2 -8351.124} C_VEL
LIN {X 0,Y 458.466,Z 522.837,A -85,B 0,C 180,E1 -8351.509,E2 -8351.509} C_VEL
LIN {X 0,Y 457.991,Z 535.711,A -85,B 0,C 180,E1 -8352.025,E2 -8352.025} C_VEL
LIN {X 0,Y 457.335,Z 548.968,A -85,B 0,C 180,E1 -8352.733,E2 -8352.733} C_VEL
LIN {X 0,Y 456.662,Z 561.279,A -85,B 0,C 180,E1 -8353.575,E2 -8353.575} C_VEL
LIN {X 0,Y 455.85,Z 573.156,A -85,B 0,C 180,E1 -8354.578,E2 -8354.578} C_VEL
LIN {X 0,Y 455.104,Z 584.004,A -85,B 0,C 180,E1 -8355.696,E2 -8355.696} C_VEL
LIN {X 0,Y 454.336,Z 594.729,A -85,B 0,C 180,E1 -8357.041,E2 -8357.041} C_VEL
LIN {X 0,Y 453.836,Z 603.568,A -85,B 0,C 180,E1 -8358.387,E2 -8358.387} C_VEL
LIN {X 0,Y 453.285,Z 612.044,A -85,B 0,C 180,E1 -8359.956,E2 -8359.956} C_VEL
LIN {X 0,Y 452.922,Z 618.869,A -85,B 0,C 180,E1 -8361.524,E2 -8361.524} C_VEL
LIN {X 0,Y 452.668,Z 623.573,A -85,B 0,C 180,E1 -8362.866,E2 -8362.866} C_VEL
LIN {X 0,Y 452.592,Z 628.451,A -85,B 0,C 180,E1 -8364.655,E2 -8364.655} C_VEL
LIN {X 0,Y 452.473,Z 631.838,A -85,B 0,C 180,E1 -8366.439,E2 -8366.439} C_VEL
LIN {X 0,Y 452.43,Z 633.839,A -85,B 0,C 180,E1 -8368.221,E2 -8368.221} C_VEL
LIN {X 0,Y 452.38,Z 634.5,A -85,B 0,C 180,E1 -8370.001,E2 -8370.001} C_VEL
LIN {X 0,Y 452.43,Z 633.834,A -85,B 0,C 180,E1 -8371.781,E2 -8371.781} C_VEL
LIN {X 0,Y 452.474,Z 631.828,A -85,B 0,C 180,E1 -8373.563,E2 -8373.563} C_VEL
LIN {X 0,Y 452.593,Z 628.439,A -85,B 0,C 180,E1 -8375.347,E2 -8375.347} C_VEL
LIN {X 0,Y 452.669,Z 623.563,A -85,B 0,C 180,E1 -8377.136,E2 -8377.136} C_VEL
LIN {X 0,Y 453.004,Z 617.047,A -85,B 0,C 180,E1 -8378.926,E2 -8378.926} C_VEL
LIN {X 0,Y 453.389,Z 609.793,A -85,B 0,C 180,E1 -8380.495,E2 -8380.495} C_VEL
LIN {X 0,Y 454.051,Z 600.809,A -85,B 0,C 180,E1 -8382.062,E2 -8382.062} C_VEL
LIN {X 0,Y 454.6,Z 591.376,A -85,B 0,C 180,E1 -8383.41,E2 -8383.41} C_VEL
LIN {X 0,Y 455.317,Z 580.932,A -85,B 0,C 180,E1 -8384.642,E2 -8384.642} C_VEL
LIN {X 0,Y 456.056,Z 569.401,A -85,B 0,C 180,E1 -8385.761,E2 -8385.761} C_VEL
LIN {X 0,Y 456.885,Z 556.604,A -85,B 0,C 180,E1 -8386.764,E2 -8386.764} C_VEL
LIN {X 0,Y 457.626,Z 543.121,A -85,B 0,C 180,E1 -8387.6,E2 -8387.6} C_VEL
LIN {X 0,Y 458.191,Z 529.811,A -85,B 0,C 180,E1 -8388.23,E2 -8388.23} C_VEL
LIN {X 0,Y 458.713,Z 515.698,A -85,B 0,C 180,E1 -8388.706,E2 -8388.706} C_VEL
LIN {X 0,Y 458.98,Z 500.681,A -85,B 0,C 180,E1 -8389.019,E2 -8389.019} C_VEL
LIN {X 0,Y 460.173,Z 394.211,A -85,B 0,C 180,E1 -8390.698,E2 -8390.698} C_VEL
LIN {X 0,Y 456.002,Z 372.387,A -85,B 0,C 180,E1 -8391.277,E2 -8391.277} C_VEL
LIN {X 0,Y 456.204,Z 367.517,A -85,B 0,C 180,E1 -8392.095,E2 -8392.095} C_VEL
LIN {X 0,Y 456.66,Z 357.918,A -85,B 0,C 180,E1 -8393.829,E2 -8393.829} C_VEL
LIN {X 0,Y 454.29,Z 345.961,A -85,B 0,C 180,E1 -8396.198,E2 -8396.198} C_VEL
LIN {X 0,Y 453.557,Z 342.683,A -85,B 0,C 180,E1 -8396.921,E2 -8396.921} C_VEL
LIN {X 0,Y 453.477,Z 342.613,A -85,B 0,C 180,E1 -8399.786,E2 -8399.786} C_VEL
LIN {X 0,Y 453.495,Z 342.619,A -85,B 0,C 180,E1 -8403.19,E2 -8403.19} C_VEL
LIN {X 0,Y 453.461,Z 342.626,A -85,B 0,C 180,E1 -8406.3,E2 -8406.3} C_VEL
LIN {X 0,Y 453.494,Z 342.62,A -85,B 0,C 180,E1 -8409.45,E2 -8409.45} C_VEL
LIN {X 0,Y 453.481,Z 342.625,A -85,B 0,C 180,E1 -8411.935,E2 -8411.935} C_VEL
LIN {X 0,Y 453.489,Z 342.622,A -85,B 0,C 180,E1 -8415.472,E2 -8415.472} C_VEL
LIN {X 0,Y 453.484,Z 342.623,A -85,B 0,C 180,E1 -8418.21,E2 -8418.21} C_VEL
LIN {X 0,Y 453.499,Z 342.619,A -85,B 0,C 180,E1 -8420.794,E2 -8420.794} C_VEL
LIN {X 0,Y 453.459,Z 342.627,A -85,B 0,C 180,E1 -8423.918,E2 -8423.918} C_VEL
LIN {X 0,Y 453.488,Z 342.623,A -85,B 0,C 180,E1 -8427.152,E2 -8427.152} C_VEL
LIN {X 0,Y 453.527,Z 342.643,A -85,B 0,C 180,E1 -8430.782,E2 -8430.782} C_VEL
LIN {X 0,Y 453.573,Z 342.939,A -85,B 0,C 180,E1 -8430.976,E2 -8430.976} C_VEL
LIN {X 0,Y 456.21,Z 353.295,A -85,B 0,C 180,E1 -8432.691,E2 -8432.691} C_VEL
LIN {X 0,Y 457.463,Z 360.328,A -85,B 0,C 180,E1 -8433.789,E2 -8433.789} C_VEL
LIN {X 0,Y 456.745,Z 380.592,A -85,B 0,C 180,E1 -8436.658,E2 -8436.658} C_VEL
LIN {X 0,Y 455.919,Z 403.983,A -85,B 0,C 180,E1 -8439.965,E2 -8439.965} C_VEL
LIN {X 0,Y 455.406,Z 420.729,A -85,B 0,C 180,E1 -8442.316,E2 -8442.316} C_VEL
LIN {X 0,Y 457.924,Z 437.883,A -85,B 0,C 180,E1 -8442.809,E2 -8442.809} C_VEL
LIN {X 0,Y 456.631,Z 520.421,A -85,B 0,C 180,E1 -8444.375,E2 -8444.375} C_VEL
LIN {X 0,Y 456.351,Z 535.503,A -85,B 0,C 180,E1 -8444.708,E2 -8444.708} C_VEL
LIN {X 0,Y 456.002,Z 548.008,A -85,B 0,C 180,E1 -8445.154,E2 -8445.154} C_VEL
LIN {X 0,Y 455.582,Z 559.367,A -85,B 0,C 180,E1 -8445.71,E2 -8445.71} C_VEL
LIN {X 0,Y 455.088,Z 571.477,A -85,B 0,C 180,E1 -8446.492,E2 -8446.492} C_VEL
LIN {X 0,Y 454.575,Z 582.019,A -85,B 0,C 180,E1 -8447.349,E2 -8447.349} C_VEL
LIN {X 0,Y 454.06,Z 592.398,A -85,B 0,C 180,E1 -8448.392,E2 -8448.392} C_VEL
LIN {X 0,Y 453.577,Z 601.405,A -85,B 0,C 180,E1 -8449.51,E2 -8449.51} C_VEL
LIN {X 0,Y 453.2,Z 610.21,A -85,B 0,C 180,E1 -8450.854,E2 -8450.854} C_VEL
LIN {X 0,Y 452.884,Z 617.251,A -85,B 0,C 180,E1 -8452.196,E2 -8452.196} C_VEL
LIN {X 0,Y 452.655,Z 623.665,A -85,B 0,C 180,E1 -8453.761,E2 -8453.761} C_VEL
LIN {X 0,Y 452.565,Z 627.847,A -85,B 0,C 180,E1 -8455.1,E2 -8455.1} C_VEL
LIN {X 0,Y 452.488,Z 630.934,A -85,B 0,C 180,E1 -8456.438,E2 -8456.438} C_VEL
LIN {X 0,Y 452.496,Z 632.437,A -85,B 0,C 180,E1 -8457.329,E2 -8457.329} C_VEL
LIN {X 0,Y 452.434,Z 633.479,A -85,B 0,C 180,E1 -8458.22,E2 -8458.22} C_VEL
LIN {X 0,Y 452.404,Z 634.119,A -85,B 0,C 180,E1 -8459.11,E2 -8459.11} C_VEL
LIN {X 0,Y 452.382,Z 634.352,A -85,B 0,C 180,E1 -8460,E2 -8460} C_VEL
LIN {X 0,Y 452.404,Z 634.124,A -85,B 0,C 180,E1 -8460.89,E2 -8460.89} C_VEL
LIN {X 0,Y 452.434,Z 633.489,A -85,B 0,C 180,E1 -8461.78,E2 -8461.78} C_VEL
LIN {X 0,Y 452.496,Z 632.453,A -85,B 0,C 180,E1 -8462.671,E2 -8462.671} C_VEL
LIN {X 0,Y 452.485,Z 630.957,A -85,B 0,C 180,E1 -8463.562,E2 -8463.562} C_VEL
LIN {X 0,Y 452.561,Z 627.88,A -85,B 0,C 180,E1 -8464.9,E2 -8464.9} C_VEL
LIN {X 0,Y 452.694,Z 622.812,A -85,B 0,C 180,E1 -8466.486,E2 -8466.486} C_VEL
LIN {X 0,Y 452.907,Z 616.244,A -85,B 0,C 180,E1 -8468.028,E2 -8468.028} C_VEL
LIN {X 0,Y 453.206,Z 608.941,A -85,B 0,C 180,E1 -8469.371,E2 -8469.371} C_VEL
LIN {X 0,Y 453.592,Z 599.85,A -85,B 0,C 180,E1 -8470.715,E2 -8470.715} C_VEL
LIN {X 0,Y 454.142,Z 589.371,A -85,B 0,C 180,E1 -8471.946,E2 -8471.946} C_VEL
LIN {X 0,Y 454.66,Z 578.473,A -85,B 0,C 180,E1 -8472.974,E2 -8472.974} C_VEL
LIN {X 0,Y 455.127,Z 566.749,A -85,B 0,C 180,E1 -8473.848,E2 -8473.848} C_VEL
LIN {X 0,Y 455.633,Z 554.147,A -85,B 0,C 180,E1 -8474.573,E2 -8474.573} C_VEL
LIN {X 0,Y 456.052,Z 540.675,A -85,B 0,C 180,E1 -8475.13,E2 -8475.13} C_VEL
LIN {X 0,Y 456.392,Z 527.332,A -85,B 0,C 180,E1 -8475.491,E2 -8475.491} C_VEL
LIN {X 0,Y 457.357,Z 437.232,A -85,B 0,C 180,E1 -8477.102,E2 -8477.102} C_VEL
LIN {X 0,Y 455.028,Z 420.918,A -85,B 0,C 180,E1 -8477.5,E2 -8477.5} C_VEL
LIN {X 0,Y 455.746,Z 399.683,A -85,B 0,C 180,E1 -8480.538,E2 -8480.538} C_VEL
LIN {X 0,Y 456.582,Z 378.568,A -85,B 0,C 180,E1 -8483.591,E2 -8483.591} C_VEL
LIN {X 0,Y 457.243,Z 360.424,A -85,B 0,C 180,E1 -8486.225,E2 -8486.225} C_VEL
LIN {X 0,Y 455.089,Z 349.498,A -85,B 0,C 180,E1 -8487.946,E2 -8487.946} C_VEL
LIN {X 0,Y 453.542,Z 342.714,A -85,B 0,C 180,E1 -8489.09,E2 -8489.09} C_VEL
LIN {X 0,Y 453.47,Z 342.625,A -85,B 0,C 180,E1 -8491.799,E2 -8491.799} C_VEL
LIN {X 0,Y 453.485,Z 342.621,A -85,B 0,C 180,E1 -8494.989,E2 -8494.989} C_VEL
LIN {X 0,Y 453.465,Z 342.628,A -85,B 0,C 180,E1 -8498.312,E2 -8498.312} C_VEL
LIN {X 0,Y 453.499,Z 342.621,A -85,B 0,C 180,E1 -8500.609,E2 -8500.609} C_VEL
LIN {X 0,Y 453.458,Z 342.618,A -85,B 0,C 180,E1 -8503.243,E2 -8503.243} C_VEL
LIN {X 0,Y 453.469,Z 342.611,A -85,B 0,C 180,E1 -8505.778,E2 -8505.778} C_VEL
LIN {X 0,Y 453.485,Z 342.624,A -85,B 0,C 180,E1 -8508.209,E2 -8508.209} C_VEL
LIN {X 0,Y 453.515,Z 342.612,A -85,B 0,C 180,E1 -8510.79,E2 -8510.79} C_VEL
LIN {X 0,Y 453.462,Z 342.62,A -85,B 0,C 180,E1 -8513.917,E2 -8513.917} C_VEL
LIN {X 0,Y 453.488,Z 342.617,A -85,B 0,C 180,E1 -8517.151,E2 -8517.151} C_VEL
LIN {X 0,Y 453.48,Z 342.603,A -85,B 0,C 180,E1 -8520.268,E2 -8520.268} C_VEL
LIN {X 0,Y 453.547,Z 342.607,A -85,B 0,C 180,E1 -8522.263,E2 -8522.263} C_VEL
LIN {X 0,Y 453.331,Z 343.095,A -85,B 0,C 180,E1 -8522.751,E2 -8522.751} C_VEL
LIN {X 0,Y 452.769,Z 344.335,A -85,B 0,C 180,E1 -8523.215,E2 -8523.215} C_VEL
LIN {X 0,Y 451.159,Z 348.196,A -85,B 0,C 180,E1 -8524.077,E2 -8524.077} C_VEL
LIN {X 0,Y 449.478,Z 354.205,A -85,B 0,C 180,E1 -8525.109,E2 -8525.109} C_VEL
LIN {X 0,Y 449.464,Z 357.575,A -85,B 0,C 180,E1 -8525.747,E2 -8525.747} C_VEL
LIN {X 0,Y 449.773,Z 361.598,A -85,B 0,C 180,E1 -8526.517,E2 -8526.517} C_VEL
LIN {X 0,Y 449.157,Z 372.336,A -85,B 0,C 180,E1 -8528.425,E2 -8528.425} C_VEL
LIN {X 0,Y 453.534,Z 394.98,A -85,B 0,C 180,E1 -8529.043,E2 -8529.043} C_VEL
LIN {X 0,Y 452.151,Z 509.154,A -85,B 0,C 180,E1 -8530.889,E2 -8530.889} C_VEL
LIN {X 0,Y 451.647,Z 523.908,A -85,B 0,C 180,E1 -8531.309,E2 -8531.309} C_VEL
LIN {X 0,Y 451.166,Z 536.789,A -85,B 0,C 180,E1 -8531.846,E2 -8531.846} C_VEL
LIN {X 0,Y 450.476,Z 549.848,A -85,B 0,C 180,E1 -8532.568,E2 -8532.568} C_VEL
LIN {X 0,Y 449.754,Z 562.091,A -85,B 0,C 180,E1 -8533.429,E2 -8533.429} C_VEL
LIN {X 0,Y 448.908,Z 573.827,A -85,B 0,C 180,E1 -8534.447,E2 -8534.447} C_VEL
LIN {X 0,Y 448.045,Z 585.537,A -85,B 0,C 180,E1 -8535.696,E2 -8535.696} C_VEL
LIN {X 0,Y 447.358,Z 594.939,A -85,B 0,C 180,E1 -8536.912,E2 -8536.912} C_VEL
LIN {X 0,Y 446.872,Z 603.278,A -85,B 0,C 180,E1 -8538.202,E2 -8538.202} C_VEL
LIN {X 0,Y 446.277,Z 611.804,A -85,B 0,C 180,E1 -8539.794,E2 -8539.794} C_VEL
LIN {X 0,Y 445.865,Z 618.676,A -85,B 0,C 180,E1 -8541.387,E2 -8541.387} C_VEL
LIN {X 0,Y 445.599,Z 623.422,A -85,B 0,C 180,E1 -8542.75,E2 -8542.75} C_VEL
LIN {X 0,Y 445.512,Z 628.333,A -85,B 0,C 180,E1 -8544.568,E2 -8544.568} C_VEL
LIN {X 0,Y 445.373,Z 631.756,A -85,B 0,C 180,E1 -8546.38,E2 -8546.38} C_VEL
LIN {X 0,Y 445.351,Z 633.794,A -85,B 0,C 180,E1 -8548.19,E2 -8548.19} C_VEL
LIN {X 0,Y 445.291,Z 634.497,A -85,B 0,C 180,E1 -8549.999,E2 -8549.999} C_VEL
LIN {X 0,Y 445.35,Z 633.874,A -85,B 0,C 180,E1 -8551.807,E2 -8551.807} C_VEL
LIN {X 0,Y 445.372,Z 631.911,A -85,B 0,C 180,E1 -8553.618,E2 -8553.618} C_VEL
LIN {X 0,Y 445.51,Z 628.557,A -85,B 0,C 180,E1 -8555.43,E2 -8555.43} C_VEL
LIN {X 0,Y 445.594,Z 623.715,A -85,B 0,C 180,E1 -8557.248,E2 -8557.248} C_VEL
LIN {X 0,Y 445.962,Z 617.24,A -85,B 0,C 180,E1 -8559.066,E2 -8559.066} C_VEL
LIN {X 0,Y 446.348,Z 610.033,A -85,B 0,C 180,E1 -8560.66,E2 -8560.66} C_VEL
LIN {X 0,Y 447.048,Z 601.119,A -85,B 0,C 180,E1 -8562.252,E2 -8562.252} C_VEL
LIN {X 0,Y 447.64,Z 591.758,A -85,B 0,C 180,E1 -8563.62,E2 -8563.62} C_VEL
LIN {X 0,Y 448.363,Z 581.389,A -85,B 0,C 180,E1 -8564.872,E2 -8564.872} C_VEL
LIN {X 0,Y 449.222,Z 569.954,A -85,B 0,C 180,E1 -8566.005,E2 -8566.005} C_VEL
LIN {X 0,Y 450.012,Z 557.283,A -85,B 0,C 180,E1 -8567.026,E2 -8567.026} C_VEL
LIN {X 0,Y 450.875,Z 543.745,A -85,B 0,C 180,E1 -8567.882,E2 -8567.882} C_VEL
LIN {X 0,Y 451.469,Z 529.998,A -85,B 0,C 180,E1 -8568.55,E2 -8568.55} C_VEL
LIN {X 0,Y 451.99,Z 516.191,A -85,B 0,C 180,E1 -8569.027,E2 -8569.027} C_VEL
LIN {X 0,Y 452.289,Z 501.948,A -85,B 0,C 180,E1 -8569.338,E2 -8569.338} C_VEL
LIN {X 0,Y 453.516,Z 394.708,A -85,B 0,C 180,E1 -8571.056,E2 -8571.056} C_VEL
LIN {X 0,Y 449.164,Z 372.315,A -85,B 0,C 180,E1 -8571.67,E2 -8571.67} C_VEL
LIN {X 0,Y 449.823,Z 359.503,A -85,B 0,C 180,E1 -8573.966,E2 -8573.966} C_VEL
LIN {X 0,Y 447.104,Z 346.205,A -85,B 0,C 180,E1 -8576.655,E2 -8576.655} C_VEL
LIN {X 0,Y 446.513,Z 343.594,A -85,B 0,C 180,E1 -8577.252,E2 -8577.252} C_VEL
LIN {X 0,Y 446.433,Z 343.486,A -85,B 0,C 180,E1 -8580.248,E2 -8580.248} C_VEL
LIN {X 0,Y 446.441,Z 343.495,A -85,B 0,C 180,E1 -8583.452,E2 -8583.452} C_VEL
LIN {X 0,Y 446.405,Z 343.502,A -85,B 0,C 180,E1 -8586.743,E2 -8586.743} C_VEL
LIN {X 0,Y 446.487,Z 343.486,A -85,B 0,C 180,E1 -8589.53,E2 -8589.53} C_VEL
LIN {X 0,Y 446.444,Z 343.497,A -85,B 0,C 180,E1 -8592.601,E2 -8592.601} C_VEL
LIN {X 0,Y 446.451,Z 343.481,A -85,B 0,C 180,E1 -8595.102,E2 -8595.102} C_VEL
LIN {X 0,Y 446.437,Z 343.497,A -85,B 0,C 180,E1 -8598.61,E2 -8598.61} C_VEL
LIN {X 0,Y 446.468,Z 343.484,A -85,B 0,C 180,E1 -8600.975,E2 -8600.975} C_VEL
LIN {X 0,Y 446.413,Z 343.497,A -85,B 0,C 180,E1 -8604.373,E2 -8604.373} C_VEL
LIN {X 0,Y 446.414,Z 343.501,A -85,B 0,C 180,E1 -8607.638,E2 -8607.638} C_VEL
LIN {X 0,Y 446.46,Z 343.466,A -85,B 0,C 180,E1 -8610.791,E2 -8610.791} C_VEL
LIN {X 0,Y 446.468,Z 343.491,A -85,B 0,C 180,E1 -8613.848,E2 -8613.848} C_VEL
LIN {X 0,Y 446.422,Z 343.499,A -85,B 0,C 180,E1 -8616.823,E2 -8616.823} C_VEL
LIN {X 0,Y 446.438,Z 343.498,A -85,B 0,C 180,E1 -8619.737,E2 -8619.737} C_VEL
LIN {X 0,Y 446.453,Z 343.493,A -85,B 0,C 180,E1 -8622.597,E2 -8622.597} C_VEL
LIN {X 0,Y 446.462,Z 343.491,A -85,B 0,C 180,E1 -8625.412,E2 -8625.412} C_VEL
LIN {X 0,Y 446.531,Z 343.483,A -85,B 0,C 180,E1 -8628.193,E2 -8628.193} C_VEL
LIN {X 0,Y 446.589,Z 343.475,A -85,B 0,C 180,E1 -8631.858,E2 -8631.858} C_VEL
LIN {X 0,Y 446.639,Z 343.472,A -85,B 0,C 180,E1 -8634.582,E2 -8634.582} C_VEL
LIN {X 0,Y 446.701,Z 343.46,A -85,B 0,C 180,E1 -8637.295,E2 -8637.295} C_VEL
LIN {X 0,Y 446.785,Z 343.453,A -85,B 0,C 180,E1 -8640,E2 -8640} C_VEL
LIN {X 0,Y 446.701,Z 343.461,A -85,B 0,C 180,E1 -8642.705,E2 -8642.705} C_VEL
LIN {X 0,Y 446.639,Z 343.472,A -85,B 0,C 180,E1 -8646.324,E2 -8646.324} C_VEL
LIN {X 0,Y 446.529,Z 343.478,A -85,B 0,C 180,E1 -8649.055,E2 -8649.055} C_VEL
LIN {X 0,Y 446.523,Z 343.49,A -85,B 0,C 180,E1 -8652.73,E2 -8652.73} C_VEL
LIN {X 0,Y 446.479,Z 343.484,A -85,B 0,C 180,E1 -8656.459,E2 -8656.459} C_VEL
LIN {X 0,Y 446.459,Z 343.491,A -85,B 0,C 180,E1 -8659.304,E2 -8659.304} C_VEL
LIN {X 0,Y 446.41,Z 343.495,A -85,B 0,C 180,E1 -8662.2,E2 -8662.2} C_VEL
LIN {X 0,Y 446.461,Z 343.491,A -85,B 0,C 180,E1 -8665.152,E2 -8665.152} C_VEL
LIN {X 0,Y 446.474,Z 343.47,A -85,B 0,C 180,E1 -8668.179,E2 -8668.179} C_VEL
LIN {X 0,Y 446.41,Z 343.494,A -85,B 0,C 180,E1 -8671.776,E2 -8671.776} C_VEL
LIN {X 0,Y 446.422,Z 343.501,A -85,B 0,C 180,E1 -8674.524,E2 -8674.524} C_VEL
LIN {X 0,Y 446.428,Z 343.478,A -85,B 0,C 180,E1 -8678.084,E2 -8678.084} C_VEL
LIN {X 0,Y 446.439,Z 343.497,A -85,B 0,C 180,E1 -8680.922,E2 -8680.922} C_VEL
LIN {X 0,Y 446.438,Z 343.49,A -85,B 0,C 180,E1 -8683.841,E2 -8683.841} C_VEL
LIN {X 0,Y 446.44,Z 343.496,A -85,B 0,C 180,E1 -8686.398,E2 -8686.398} C_VEL
LIN {X 0,Y 446.463,Z 343.488,A -85,B 0,C 180,E1 -8689.806,E2 -8689.806} C_VEL
LIN {X 0,Y 446.429,Z 343.504,A -85,B 0,C 180,E1 -8692.125,E2 -8692.125} C_VEL
LIN {X 0,Y 446.426,Z 343.5,A -85,B 0,C 180,E1 -8695.478,E2 -8695.478} C_VEL
LIN {X 0,Y 446.427,Z 343.501,A -85,B 0,C 180,E1 -8698.702,E2 -8698.702} C_VEL
LIN {X 0,Y 446.481,Z 343.479,A -85,B 0,C 180,E1 -8701.823,E2 -8701.823} C_VEL
LIN {X 0,Y 446.528,Z 343.713,A -85,B 0,C 180,E1 -8702.844,E2 -8702.844} C_VEL
LIN {X 0,Y 448.999,Z 355.136,A -85,B 0,C 180,E1 -8705.21,E2 -8705.21} C_VEL
LIN {X 0,Y 449.856,Z 360.57,A -85,B 0,C 180,E1 -8706.28,E2 -8706.28} C_VEL
LIN {X 0,Y 449.13,Z 372.32,A -85,B 0,C 180,E1 -8708.373,E2 -8708.373} C_VEL
LIN {X 0,Y 453.564,Z 395.384,A -85,B 0,C 180,E1 -8709.003,E2 -8709.003} C_VEL
LIN {X 0,Y 452.176,Z 508.774,A -85,B 0,C 180,E1 -8710.833,E2 -8710.833} C_VEL
LIN {X 0,Y 451.75,Z 522.921,A -85,B 0,C 180,E1 -8711.227,E2 -8711.227} C_VEL
LIN {X 0,Y 451.249,Z 535.477,A -85,B 0,C 180,E1 -8711.735,E2 -8711.735} C_VEL
LIN {X 0,Y 450.543,Z 549.232,A -85,B 0,C 180,E1 -8712.482,E2 -8712.482} C_VEL
LIN {X 0,Y 449.837,Z 561.283,A -85,B 0,C 180,E1 -8713.318,E2 -8713.318} C_VEL
LIN {X 0,Y 448.992,Z 573.159,A -85,B 0,C 180,E1 -8714.336,E2 -8714.336} C_VEL
LIN {X 0,Y 448.17,Z 584.006,A -85,B 0,C 180,E1 -8715.47,E2 -8715.47} C_VEL
LIN {X 0,Y 447.44,Z 594.206,A -85,B 0,C 180,E1 -8716.763,E2 -8716.763} C_VEL
LIN {X 0,Y 446.864,Z 603.57,A -85,B 0,C 180,E1 -8718.204,E2 -8718.204} C_VEL
LIN {X 0,Y 446.255,Z 612.046,A -85,B 0,C 180,E1 -8719.796,E2 -8719.796} C_VEL
LIN {X 0,Y 445.855,Z 618.87,A -85,B 0,C 180,E1 -8721.389,E2 -8721.389} C_VEL
LIN {X 0,Y 445.594,Z 623.574,A -85,B 0,C 180,E1 -8722.752,E2 -8722.752} C_VEL
LIN {X 0,Y 445.509,Z 628.451,A -85,B 0,C 180,E1 -8724.57,E2 -8724.57} C_VEL
LIN {X 0,Y 445.372,Z 631.839,A -85,B 0,C 180,E1 -8726.382,E2 -8726.382} C_VEL
LIN {X 0,Y 445.349,Z 633.839,A -85,B 0,C 180,E1 -8728.193,E2 -8728.193} C_VEL
LIN {X 0,Y 445.29,Z 634.5,A -85,B 0,C 180,E1 -8730.001,E2 -8730.001} C_VEL
LIN {X 0,Y 445.349,Z 633.834,A -85,B 0,C 180,E1 -8731.81,E2 -8731.81} C_VEL
LIN {X 0,Y 445.372,Z 631.828,A -85,B 0,C 180,E1 -8733.62,E2 -8733.62} C_VEL
LIN {X 0,Y 445.51,Z 628.438,A -85,B 0,C 180,E1 -8735.432,E2 -8735.432} C_VEL
LIN {X 0,Y 445.595,Z 623.562,A -85,B 0,C 180,E1 -8737.25,E2 -8737.25} C_VEL
LIN {X 0,Y 445.964,Z 617.045,A -85,B 0,C 180,E1 -8739.068,E2 -8739.068} C_VEL
